// TIA Portal project "СУК 3.2 РАЕС-1.2 v1.1_20261002_1325" (V20)

(* hardware
DEVICE "S7-1500/ET200MP station_1"  S7-1500 station
   slot 0: "Rail_0"  Rack  6ES7 590-1***0-0AA0
   slot 1: "A1_1"  CPU 1515-2 PN  6ES7 515-2AN03-0AB0  V3.0
      slot 3: "CPU display_1"  6ES7591-1BA00-0AA0
      slot 32768: "PROFINET interface_1"  X1
         slot 32769: "Port_1"  X1 P1
         slot 32770: "Port_2"  X1 P2
      slot 33024: "PROFINET interface_2"  X2
         slot 33025: "Port_1"  X2 P1
      slot 34817: "Virtual CP interface port_1"  Virtual CP interface port  Virtual CP interface port
   slot 2: "A1_2"  DI 32x24VDC HF  6ES7 521-1BL00-0AB0  V2.2
   slot 3: "A1_3"  DI 32x24VDC HF  6ES7 521-1BL00-0AB0  V2.2
   slot 4: "A1_4"  AI 8xU/I HF  6ES7 531-7NF00-0AB0  V1.2
   slot 5: "A1_5"  DQ 16x24VDC/0.5A HF  6ES7 522-1BH01-0AB0  V1.0
DEVICE "A1_0"  TP700 Comfort
   slot 0: "A1_0"  TP700 Comfort  6AV2 124-0GC01-0AX0  17.0.0.0
   slot 1: "HMI_RT_1"  TP700 Comfort  6AV2 124-0GC01-0AX0  17.0.0.0
   slot 5: "A1_0.IE_CP_1"  PROFINET Interface  17.0.0.0
      slot 1: "PROFINET Interface_1"  PROFINET Interface
         slot 1: "Port_1"  Port
         slot 2: "Port_2"  Port
   slot 7: "A1_0.MPI/DP_CP_1"  MPI/DP Interface  17.0.0.0
DEVICE "SCALANCE XC-200"  SCALANCE X-Station
   slot 0: "SCALANCE X rack"  Rail
   slot 0: "A1.6"  SCALANCE XC208  6GK5 208-0BA00-2AC2  V4.4
DEVICE "GSD device_1"  GSD.Device.PN
   slot 0: "Rack"  Rack  V1.0
   slot 0: "1BR"  Multiturn 30 Bit V2.x  6FX2001-5*N25  V2.2.x
      slot 0: "MC-Encoder Multiturn 30 Bit"  MC-Encoder Multiturn 30 Bit
      slot 1: "PN-IO"  PN-IO
         slot 1: "Port 1"  Port 1
         slot 2: "Port 2"  Port 2
      slot 1: "EO Encoder Multiturn V2.x_1"  EO Encoder Multiturn V2.x
         slot 0: "Module Access Point"  Module Access Point
   slot 1: "Standard Telegram 89, PZD3/5"  Standard Telegram 89, PZD3/5
DEVICE "GSD device_2"  GSD.Device.PN
   slot 0: "Rack"  Rack  V1.0
   slot 0: "3BR"  Multiturn 30 Bit V2.x  6FX2001-5*N25  V2.2.x
      slot 0: "MC-Encoder Multiturn 30 Bit"  MC-Encoder Multiturn 30 Bit
      slot 1: "PN-IO"  PN-IO
         slot 1: "Port 1"  Port 1
         slot 2: "Port 2"  Port 2
      slot 1: "EO Encoder Multiturn V2.x_1"  EO Encoder Multiturn V2.x
         slot 0: "Module Access Point"  Module Access Point
   slot 1: "Standard Telegram 89, PZD3/5"  Standard Telegram 89, PZD3/5
DEVICE "GSD device_3"  GSD.Device.PN
   slot 0: "Rack"  Rack  V1.0
   slot 0: "4BR1"  Multiturn 30 Bit V2.x  6FX2001-5*N25  V2.2.x
      slot 0: "MC-Encoder Multiturn 30 Bit"  MC-Encoder Multiturn 30 Bit
      slot 1: "PN-IO"  PN-IO
         slot 1: "Port 1"  Port 1
         slot 2: "Port 2"  Port 2
      slot 1: "EO Encoder Multiturn V2.x_1"  EO Encoder Multiturn V2.x
         slot 0: "Module Access Point"  Module Access Point
   slot 1: "Standard Telegram 89, PZD3/5"  Standard Telegram 89, PZD3/5
DEVICE "GSD device_4"  GSD.Device.PN
   slot 0: "Rack"  Rack  V1.0
   slot 0: "4BR2"  Multiturn 30 Bit V2.x  6FX2001-5*N25  V2.2.x
      slot 0: "MC-Encoder Multiturn 30 Bit"  MC-Encoder Multiturn 30 Bit
      slot 1: "PN-IO"  PN-IO
         slot 1: "Port 1"  Port 1
         slot 2: "Port 2"  Port 2
      slot 1: "EO Encoder Multiturn V2.x_1"  EO Encoder Multiturn V2.x
         slot 0: "Module Access Point"  Module Access Point
   slot 1: "Standard Telegram 89, PZD3/5"  Standard Telegram 89, PZD3/5
DEVICE "SINAMICS S_1"  SINAMICS S120
   slot 0: "Drive unit_1"  S120 CU320-2 PN  6SL3040-1MA01-0Axx  V5.1
      slot 1: "PROFINET interface"  PROFINET
      slot 3: "Ethernet commissioning interface"  LAN
   slot 0: "U1"  S120 CU320-2 PN
   slot 1: "1UZ1"  PM
      slot 10: "Control Unit Adapter_1"  1UZ1  6SL3040-0PA00-0Axx
      slot 200: "Power Module_1"  1UZ1  6SL3210-1PE21-4UL0
      slot 1000: "1M1"  1UZ1  XMxxxxx-xxxxx-xxxx
   slot 2: "3UZ1"  PM
      slot 10: "Control Unit Adapter_1"  3UZ1  6SL3040-0PA00-0Axx
      slot 200: "Power Module_2"  3UZ1  6SL3210-1PE14-3UL1
      slot 1000: "3M1"  3UZ1  XMxxxxx-xxxxx-xxxx
   slot 3: "4UZ1"  PM
      slot 10: "Control Unit Adapter_1"  4UZ1  6SL3040-0PA00-0Axx
      slot 200: "Power Module_3"  4UZ1  6SL3210-1PE14-3UL1
      slot 1000: "4M1"  4UZ1  XMxxxxx-xxxxx-xxxx
   slot 4: "4UZ2"  PM
      slot 10: "Control Unit Adapter_1"  4UZ2  6SL3040-0PA00-0Axx
      slot 200: "Power Module_4"  4UZ2  6SL3210-1PE14-3UL1
      slot 1000: "4M2"  4UZ2  XMxxxxx-xxxxx-xxxx
*)

// ===== PLC "A1_1"  CPU 1515-2 PN =====

VAR_GLOBAL   // PLC tag table "Default tag table"
   "xInitMerker" AT %M3.0 : Bool;   // Ознака ініціалізація панелі
   "TestReset" AT %M0.0 : Bool;
   "Clock_Byte" AT %MB0 : Byte;
   "Clock_10Hz" AT %M0.0 : Bool;
   "Clock_5Hz" AT %M0.1 : Bool;
   "Clock_2.5Hz" AT %M0.2 : Bool;
   "Clock_2Hz" AT %M0.3 : Bool;
   "Clock_1.25Hz" AT %M0.4 : Bool;
   "Clock_1Hz" AT %M0.5 : Bool;
   "Clock_0.625Hz" AT %M0.6 : Bool;
   "Clock_0.5Hz" AT %M0.7 : Bool;
END_VAR

VAR_GLOBAL   // PLC tag table "IO_Tags"
   "6KM1" AT %I0.0 : Bool;   // Лінійний контактор включений
   "6KM2" AT %I0.1 : Bool;   // Контактор кіл управління 220В, 50Гц включений
   "6KV" AT %I0.2 : Bool;   // Контроль напруги введення, 380В, 50Гц
   "6SF5" AT %I0.3 : Bool;   // Вимикач кіл живлення обігріву 220В, 50Гц
   "6QF2" AT %I0.4 : Bool;   // Захист кіл гальм
   "6QF3" AT %I0.5 : Bool;   // Вимикач трансформатора 6Т1, 380В, 50Гц
   "6QF4" AT %I0.6 : Bool;   // Вимикач вторинних кіл трансформатора 6Т1, 380В, 50Гц
   "6SF1" AT %I0.7 : Bool;   // Вимикач живлення 6KV, 380В, 50Гц
   "6SF2" AT %I1.0 : Bool;   // Ввідний пристрій. Вимикач кіл управління 220В, 50Гц
   "6SF4" AT %I1.1 : Bool;   // Ввідний пристрій. Вимикач кіл живлення ОВП, 220В, 50Гц
   "6K3" AT %I1.2 : Bool;   // Ввідний пристрій. Команда на включення лінійного контактора з пульта
   "9QF2" AT %I1.3 : Bool;   // Вимикач трансформатора 9Т1, 380В, 50Гц
   "9QF3" AT %I1.4 : Bool;   // Вимикач ремонтного освітлення, 12В, 50Гц
   "9QF4" AT %I1.5 : Bool;   // Вимикач власних потреб шафа, 220В, 50Гц
   "9K2" AT %I1.6 : Bool;   // Контроль підігріву шафи SU1
   "9K3" AT %I1.7 : Bool;   // Сейсмодатчик
   "S1_Up" AT %I2.0 : Bool;   // Механізм підйому. Підйом 1-а швидкість
   "S1_Down" AT %I2.1 : Bool;   // Механізм підйому. Опускання 1-а швидкість
   "S1_Forward" AT %I2.2 : Bool;   // Механізм пересування візка. Вперед 1-а швидкість
   "S1_Backward" AT %I2.3 : Bool;   // Механізм пересування візка. Назад 1-а швидкість
   "S1_Left" AT %I2.4 : Bool;   // Механізм пересування крана. Вліво 1-а швидкість
   "S1_Right" AT %I2.5 : Bool;   // Механізм пересування крана. Управо 1-а швидкість
   "S2_Speed" AT %I2.6 : Bool;   // Перемикач 2-а швидкість
   "Bell" AT %I2.7 : Bool;   // Включення дзвінка
   "1BV" AT %I3.1 : Bool;   // Контроль обертання барабану
   "1BM1_Up" AT %I3.2 : Bool;   // Контроль роботи механізма підйому
   "1BM1_Brake" AT %I3.3 : Bool;   // Контроль зносу гальма механізму підйому
   "1K41" AT %I3.4 : Bool;   // Дозвіл роботи механізмупідйому. (РП роз'єданий з приводом)
   "4QF1" AT %I3.5 : Bool;   // Механізм пересування крана. Захист кіл гальм
   "4KT1" AT %I3.6 : Bool;   // Механізм пересування крана. Температурний захист двигуна 4M1
   "4KT2" AT %I3.7 : Bool;   // Механізм пересування крана. Температурний захист двигуна 4M2
   "1BT1" AT %I4.0 : Bool;   // Механізм підйому. Термозахист гальмівного резистора
   "1K1" AT %I4.1 : Bool;   // Механізм підйому. Дозвіл нормальної швидкості. Рух вгору
   "1K2" AT %I4.2 : Bool;   // Механізм підйому. Дозвіл нормальної швидкості. Рух вниз
   "1K3" AT %I4.3 : Bool;   // Механізм підйому. Дозвіл роботи. Рух вгору
   "1K4" AT %I4.4 : Bool;   // Механізм підйому. Дозвіл роботи. Рух вниз
   "1K11" AT %I4.5 : Bool;   // Механізм підйому. Перевищення номінального вантажу 115%
   "1K12" AT %I4.6 : Bool;   // Механізм підйому. Ослаблення канатів
   "1KT" AT %I4.7 : Bool;   // Механізм підйому. Температурний захист двигуна
   "1K21" AT %I5.0 : Bool;   // Механізм підйому. Вимикачі кінцеві на гальмі 1YB1. Гальмо розгальмоване
   "1K22" AT %I5.1 : Bool;   // Механізм підйому. Вимикачі кінцеві на гальмі 1YB1. Гальмо загальмоване
   "1K23" AT %I5.2 : Bool;   // Механізм підйому. Вимикачі кінцеві на гальмі 1YB1. Товщина гальмівних наладок в нормі
   "1K31" AT %I5.3 : Bool;   // Механізм підйому. Вимикачі кінцеві на гальмі 1YB2. Гальмо розгальмоване
   "1K32" AT %I5.4 : Bool;   // Механізм підйому. Вимикачі кінцеві на гальмі 1YB2. Гальмо загальмоване
   "1K33" AT %I5.5 : Bool;   // Механізм підйому. Вимикачі кінцеві на гальмі 1YB2. Дозвіл роботи (MPP роз'єднаний з гальмом)
   "1QF1" AT %I5.6 : Bool;   // Механізм підйому. Захист випрямляча гальма 1YB1
   "1QF2" AT %I5.7 : Bool;   // Механізм підйому. Захист випрямляча гальма 1YB2
   "3BT1" AT %I6.0 : Bool;   // Механізм пересування візка. Термозахист гальмівного резистора
   "3K1" AT %I6.1 : Bool;   // Механізм пересування візка. Дозвіл нормальної швидкості. Рух вперед
   "3K2" AT %I6.2 : Bool;   // Механізм пересування візка. Дозвіл роботи. Рух вперед
   "3K3" AT %I6.3 : Bool;   // Механізм пересування візка. Дозвіл нормальної швидкості. Рух назад
   "3K4" AT %I6.4 : Bool;   // Механізм пересування візка. Дозвіл роботи. Рух назад
   "3K41" AT %I6.5 : Bool;   // Механізм пересування візка. Дозвіл роботи (РП роз'єднан з приводом)
   "3KT" AT %I6.6 : Bool;   // Механізм пересування візка. Температурний захист двигуна
   "4K5" AT %I6.7 : Bool;   // Механізм пересування крана. Дозвіл роботи з будь-якої зі сторін від колони
   "4BT1" AT %I7.0 : Bool;   // Механізм пересування крана. Термозахист гальмівного резистора 4RT1
   "4BT2" AT %I7.1 : Bool;   // Механізм пересування крана. Термозахист гальмівного резистора 4RT2
   "4K1" AT %I7.2 : Bool;   // Механізм пересування крана. Дозвіл нормальної швидкості. Рух вліво
   "4K2" AT %I7.3 : Bool;   // Механізм пересування крана. Дозвіл нормальної швидкості. Рух управо
   "4K3" AT %I7.4 : Bool;   // Механізм пересування крана. Дозвіл роботи. Рух вліво
   "4K4" AT %I7.5 : Bool;   // Механізм пересування крана. Дозвіл роботи. Рух управо
   "4K41" AT %I7.6 : Bool;   // Механізм пересування крана. Дозвіл роботи (РП роз'єднан з приводом). 4SQ41
   "4K42" AT %I7.7 : Bool;   // Механізм пересування крана. Дозвіл роботи (РП роз'єднан з приводом). 4SQ42
   "1KM1" AT %Q0.0 : Bool;   // Включення рабочого гальма підйому
   "1KM2" AT %Q0.1 : Bool;   // Включення вбудованого гальма підйому
   "1KM3" AT %Q0.2 : Bool;   // Включення аварійного гальма підйому
   "3KM1" AT %Q0.3 : Bool;   // Включення рабочого гальма пересування візка
   "4KM1" AT %Q0.4 : Bool;   // Включення рабочих гальм пересування крана
   "6K1" AT %Q0.5 : Bool;   // Дозвіл включення лінійного контактора
   "6K2" AT %Q0.6 : Bool;   // Вимкнення лінійного контактора
   "9K1" AT %Q0.7 : Bool;   // Включення дзвінка
   "S1_1HL" AT %Q1.2 : Bool;   // Лампа. Готовність приводу підйому
   "S1_3HL" AT %Q1.3 : Bool;   // Лампа. Готовність приводу пересування візка
   "S1_4HL" AT %Q1.4 : Bool;   // Лампа. Готовність приводу пересування крана
   "S1_6HL1" AT %Q1.5 : Bool;   // Лампа. Лінійний контактор увімкнено
   "S1_6HL2" AT %Q1.6 : Bool;   // Лампа. Вхідна напруга не в нормі
   "1A1" AT %IW8 : Int;   // Контроль крутного моменту двигуна підйома
   "I3_0" AT %I3.0 : Bool;   // Резерв
   "IW10" AT %IW10 : Int;   // Резерв
   "IW12" AT %IW12 : Int;   // Резерв
   "IW14" AT %IW14 : Int;   // Резерв
   "IW16" AT %IW16 : Int;   // Резерв
   "IW18" AT %IW18 : Int;   // Резерв
   "IW20" AT %IW20 : Int;   // Резерв
   "IW22" AT %IW22 : Int;   // Резерв
   "Q1_0" AT %Q1.0 : Bool;   // Резерв
   "Q1_1" AT %Q1.1 : Bool;   // Резерв
   "Q1_7" AT %Q1.7 : Bool;   // Резерв
END_VAR

TYPE "udtMovePerm"
   STRUCT
      Upward : Bool;   // Дозвіл роботи. Рух вгору
      Downward : Bool;   // Дозвіл роботи. Рух вниз
      Forward : Bool;   // Дозвіл роботи. Рух вперед
      Backward : Bool;   // Дозвіл роботи. Рух назад
      Left : Bool;   // Дозвіл роботи. Рух вліво
      Right : Bool;   // Дозвіл роботи. Рух управо
      No_Pillar : Bool;   // Дозвіл роботи. Збудь-якої зі сторін від колони
   END_STRUCT;
END_TYPE

TYPE "DigICfg"
   STRUCT
      VRaw : Bool;   // RAW value
      Val : Bool;   // Value
      INV : Bool;   // Inverse raw value
      SVal : Bool;   // Value for simulation
      SML : Bool;   // Output value is simulated
      Text : WString;   // Tag name
      Chanal : WString;   // Chanal
   END_STRUCT;
END_TYPE

TYPE "udtMDM"
   STRUCT
      LM_WP_disconn_brake : Bool;   // Механізм підйому. Вимикачі кінцеві на гальмі 1YB2. Дозвіл роботи (MPP роз'єднаний з гальмом)
      LM_WP_disconn_drive : Bool;   // Механізм підйому. РП роз'єднаний з приводом
      TM_WP_disconn_drive : Bool;   // Механізм пересування візка. Дозвіл роботи (РП роз'єднан з приводом)
      CM_WP_disconn_drive_1 : Bool;   // Механізм пересування крана. Дозвіл роботи (РП роз'єднан з приводом). 4SQ41
      CM_WP_disconn_drive_2 : Bool;   // Механізм пересування крана. Дозвіл роботи (РП роз'єднан з приводом). 4SQ42
   END_STRUCT;
END_TYPE

TYPE "AnICfg"
   STRUCT
      VRaw : Int;   // Raw value (from input channel)
      LORaw : Int;   // Raw value LO limit
      HIRaw : Int;   // RAW value HI limit
      Val : Real;   // Output value
      LOEng : Real;   // Engineering (scaled) minimum value
      HIEng : Real;   // Engineering (scaled) maximum value
      FVal : Real;   // Filtered value
      PhyVal : Real;   // Physical value (mA)
      LOSP : Real;   // LO setpoint
      LOLOSP : Real;   // LO-LO setpoint
      HISP : Real;   // HI setpoint
      HIHISP : Real;   // HI-HI setpoint
      Hyst : Real;   // Hysteresis in real units
      SimVal : Real;   // Value for simulation
      LOEn : Bool;   // LO warning enabled
      LOLOEn : Bool;   // LO-LO Alarm enabled
      HIEn : Bool;   // HI warning enabled
      HIHIEn : Bool;   // HI-HI Alarm enabled
      LO : Bool;   // Low level is reached
      LOLO : Bool;   // Low Low level is reached
      HI : Bool;   // High level is reached
      HIHI : Bool;   // High High level is reached
      SML : Bool;   // Output value is simulated
      Reset : Bool;   // Reset
      STS : Int;   // Status
      T_FLTR : Int;   // Filtering time, x0.01 seconds
      Text : WString;   // Tag name
      Chanal : WString;   // Chanal
   END_STRUCT;
END_TYPE

TYPE "udtRemCtrl"
   STRUCT
      Btn_Up : Bool;   // 1SB1 Підйом 1 швидкість
      Btn_Down : Bool;   // 1SB2 Опускання 1 швидкість
      Btn_Fwd : Bool;   // 3SB1 Вперед 1-а швидкість
      Btn_Bwd : Bool;   // 3SB2 Назад 1-а швидкість
      Btn_Left : Bool;   // 4SB1 Управо 1-а швидкість
      Btn_Right : Bool;   // 4SB2 Вліво 1-а швидкість
      Btn_ScndSpeed : Bool;   // SB1 2 швидкість
      Btn_Bell : Bool;   // 9SB1 Включення дзвінка
   END_STRUCT;
END_TYPE

TYPE "DigOCfg"
   STRUCT
      VRaw : Bool;
      Val : Bool;
      SVal : Bool;
      SML : Bool;
      Text : WString;
      Chanal : WString;
   END_STRUCT;
END_TYPE

TYPE "udtSpeedPerm"
   STRUCT
      Speed_normal_Up : Bool;   // Дозвіл ном. швидкості вгору
      Speed_normal_Down : Bool;   // Дозвіл ном. швидкості вниз
      Speed_normal_Fwd : Bool;   // Дозвіл ном. швидкості вперед
      Speed_normal_Bwd : Bool;   // Дозвіл ном. швидкості назад
      Speed_normal_Left : Bool;   // Дозвіл ном. швидкості вліво
      Speed_normal_Right : Bool;   // Дозвіл ном. швидкості вправо
   END_STRUCT;
END_TYPE

// folder: Drives

TYPE "UDT_S120_Tel220_In"
   STRUCT
      ZSW1_BM : Word := W#16#0000;   // PZD1 Основне статусне слово ПЧ
      NIST_A : Int := 0;   // PZD2 Фактична швидкість
      IAIST : Int := 0;   // PZD3 Фактичний струм
      MIST : Int := 0;   // PZD4 Фактичний момент
      WARN_CODE : Word := W#16#0000;   // PZD5 Код попередження ПЧ
      FAULT_CODE : Word := W#16#0000;   // PZD6 Код аварії ПЧ
      ZSW2_BM : Word := W#16#0000;   // PZD7 Додаткове статусне слово ПЧ
      NSET_FB : Int := 0;   // PZD8 Зворотний зв'язок по завданню швидкості з ПЧ
      P_ACT : Int := 0;   // PZD9 Поточна активна потужність ПЧ
      BRAKE_STATUS : Word := W#16#0000;   // PZD10 Статус гальма з ПЧ, параметр r1229
   END_STRUCT;
END_TYPE

TYPE "UDT_S120_Tel220_Out"
   STRUCT
      STW1_BM : Word := W#16#0000;   // PZD1 Основне керуюче слово ПЧ
      NSOLL_B : DInt := 0;   // PZD2-PZD3 Завдання швидкості (32 Bits) / PZD2 Завдання швидкості
      STW2_BM : Word := W#16#0000;   // PZD4 Додаткове керуюче слово ПЧ / PZD3 Додаткове керуюче слово ПЧ
      M_ADD : Int := 0;   // PZD5 Додаткове завдання моменту / PZD4 Додаткове завдання моменту
      M_LIM : Int := 0;   // PZD6 Обмеження моменту / PZD5 Обмеження моменту
      USER_1 : Word := W#16#0000;   // PZD7 Резерв / сигнал прикладної логіки / PZD6 Резерв / сигнал прикладної логіки
      USER_2 : Word := W#16#0000;   // PZD8 Резерв / сигнал прикладної логіки / PZD7 Резерв / сигнал прикладної логіки
      USER_3 : Word := W#16#0000;   // PZD9 Резерв / сигнал прикладної логіки / PZD8 Резерв / сигнал прикладної логіки
      USER_4 : Word := W#16#0000;   // PZD10 Резерв / сигнал прикладної логіки / PZD9 Резерв / сигнал прикладної логіки
   END_STRUCT;
END_TYPE

TYPE "UDT_S120_BrakeStatus"
   STRUCT
      CommandOpenBrake : Bool := FALSE;   // Біт 01: команда відкрити гальмо, постійний сигнал
      PulseEnableExtendedBrakeControl : Bool := FALSE;   // Біт 03: імпульс дозволу розширеного керування гальмом
      BrakeDoesNotOpen : Bool := FALSE;   // Біт 04: гальмо не відкривається
      BrakeDoesNotClose : Bool := FALSE;   // Біт 05: гальмо не закривається
      BrakeThresholdExceeded : Bool := FALSE;   // Біт 06: перевищено поріг гальма
      BrakeThresholdUndershot : Bool := FALSE;   // Біт 07: значення нижче порогу гальма
      BrakeMonitoringTimeExpired : Bool := FALSE;   // Біт 08: перевищено час контролю гальма
      PulseEnableRequestMissing : Bool := FALSE;   // Біт 09: відсутній запит дозволу імпульсу / керування заблоковано
      BrakeOrLogicResult : Bool := FALSE;   // Біт 10: результат логіки OR для гальма
      BrakeAndLogicResult : Bool := FALSE;   // Біт 11: результат логіки AND для гальма
   END_STRUCT;
END_TYPE

TYPE "UDT_HMI_WordBits"
   STRUCT
      Bit00 : Bool := FALSE;   // Біт 00
      Bit01 : Bool := FALSE;   // Біт 01
      Bit02 : Bool := FALSE;   // Біт 02
      Bit03 : Bool := FALSE;   // Біт 03
      Bit04 : Bool := FALSE;   // Біт 04
      Bit05 : Bool := FALSE;   // Біт 05
      Bit06 : Bool := FALSE;   // Біт 06
      Bit07 : Bool := FALSE;   // Біт 07
      Bit08 : Bool := FALSE;   // Біт 08
      Bit09 : Bool := FALSE;   // Біт 09
      Bit10 : Bool := FALSE;   // Біт 10
      Bit11 : Bool := FALSE;   // Біт 11
      Bit12 : Bool := FALSE;   // Біт 12
      Bit13 : Bool := FALSE;   // Біт 13
      Bit14 : Bool := FALSE;   // Біт 14
      Bit15 : Bool := FALSE;   // Біт 15
   END_STRUCT;
END_TYPE

TYPE "UDT_HMI_S120_STW1"
   STRUCT
      OnOff1 : Bool := FALSE;   // Біт 00: ON / OFF1
      NoCoastStop : Bool := FALSE;   // Біт 01: OFF2 не активний
      NoQuickStop : Bool := FALSE;   // Біт 02: OFF3 / Quick Stop не активний
      EnableOperation : Bool := FALSE;   // Біт 03: дозвіл роботи ПЧ
      RampGeneratorEnable : Bool := FALSE;   // Біт 04: дозвіл генератора рампи
      RampGeneratorContinue : Bool := FALSE;   // Біт 05: продовження роботи генератора рампи
      SetpointEnable : Bool := FALSE;   // Біт 06: дозвіл завдання швидкості
      FaultAcknowledge : Bool := FALSE;   // Біт 07: квітування аварії ПЧ
      Reserved08 : Bool := FALSE;   // Біт 08: резерв / залежить від параметрування
      Reserved09 : Bool := FALSE;   // Біт 09: резерв / залежить від параметрування
      ControlByPLC : Bool := FALSE;   // Біт 10: керування від PLC
      Reserved11 : Bool := FALSE;   // Біт 11: резерв / залежить від параметрування
      Reserved12 : Bool := FALSE;   // Біт 12: резерв / залежить від параметрування
      Reserved13 : Bool := FALSE;   // Біт 13: резерв / залежить від параметрування
      Reserved14 : Bool := FALSE;   // Біт 14: резерв / залежить від параметрування
      Reserved15 : Bool := FALSE;   // Біт 15: резерв / залежить від параметрування
   END_STRUCT;
END_TYPE

TYPE "UDT_HMI_S120_ZSW1"
   STRUCT
      ReadyToSwitchOn : Bool := FALSE;   // Біт 00: ПЧ готовий до вмикання
      ReadyToOperate : Bool := FALSE;   // Біт 01: ПЧ готовий до роботи
      OperationEnabled : Bool := FALSE;   // Біт 02: робота ПЧ дозволена
      FaultActive : Bool := FALSE;   // Біт 03: активна аварія ПЧ
      NoCoastStopActive : Bool := FALSE;   // Біт 04: OFF2 не активний
      NoQuickStopActive : Bool := FALSE;   // Біт 05: OFF3 / Quick Stop не активний
      SwitchingOnInhibit : Bool := FALSE;   // Біт 06: активна заборона вмикання
      WarningActive : Bool := FALSE;   // Біт 07: активне попередження ПЧ
      SpeedErrorInTolerance : Bool := FALSE;   // Біт 08: відхилення швидкості в межах допуску / залежить від параметрування
      ControlRequested : Bool := FALSE;   // Біт 09: ПЧ запитує керування від PLC
      SetpointReached : Bool := FALSE;   // Біт 10: завдання досягнуто / залежить від параметрування
      InternalLimitActive : Bool := FALSE;   // Біт 11: активне внутрішнє обмеження
      Reserved12 : Bool := FALSE;   // Біт 12: резерв / залежить від параметрування
      Reserved13 : Bool := FALSE;   // Біт 13: резерв / залежить від параметрування
      Reserved14 : Bool := FALSE;   // Біт 14: резерв / залежить від параметрування
      Reserved15 : Bool := FALSE;   // Біт 15: резерв / залежить від параметрування
   END_STRUCT;
END_TYPE

TYPE "UDT_HMI_S120_BrakeStatus"
   STRUCT
      RawWord : Word := W#16#0000;   // Сире слово статусу гальма з ПЧ
      Bit00 : Bool := FALSE;   // Біт 00: резерв / не використовується
      CommandOpenBrake : Bool := FALSE;   // Біт 01: команда відкрити гальмо
      Bit02 : Bool := FALSE;   // Біт 02: резерв / не використовується
      PulseEnableExtendedBrakeControl : Bool := FALSE;   // Біт 03: імпульс дозволу розширеного керування гальмом
      BrakeDoesNotOpen : Bool := FALSE;   // Біт 04: гальмо не відкривається
      BrakeDoesNotClose : Bool := FALSE;   // Біт 05: гальмо не закривається
      BrakeThresholdExceeded : Bool := FALSE;   // Біт 06: перевищено поріг гальма
      BrakeThresholdUndershot : Bool := FALSE;   // Біт 07: значення нижче порогу гальма
      BrakeMonitoringTimeExpired : Bool := FALSE;   // Біт 08: перевищено час контролю гальма
      PulseEnableRequestMissing : Bool := FALSE;   // Біт 09: відсутній запит дозволу імпульсу / керування заблоковано
      BrakeOrLogicResult : Bool := FALSE;   // Біт 10: результат логіки OR для гальма
      BrakeAndLogicResult : Bool := FALSE;   // Біт 11: результат логіки AND для гальма
      Bit12 : Bool := FALSE;   // Біт 12: резерв / не використовується
      Bit13 : Bool := FALSE;   // Біт 13: резерв / не використовується
      Bit14 : Bool := FALSE;   // Біт 14: резерв / не використовується
      Bit15 : Bool := FALSE;   // Біт 15: резерв / не використовується
   END_STRUCT;
END_TYPE

TYPE "UDT_HMI_S120_RawTelegram"
   STRUCT
      STW1_BM : Word := W#16#0000;   // PZD1 PLC -> ПЧ: основне керуюче слово
      NSOLL_B : DInt := 0;   // PZD2-PZD3 PLC -> ПЧ: завдання швидкості (32 Bits) / PZD2 PLC -> ПЧ: завдання швидкості
      STW2_BM : Word := W#16#0000;   // PZD4 PLC -> ПЧ: додаткове керуюче слово / PZD3 PLC -> ПЧ: додаткове керуюче слово
      M_ADD : Int := 0;   // PZD5 PLC -> ПЧ: додаткове завдання моменту / PZD4 PLC -> ПЧ: додаткове завдання моменту
      M_LIM : Int := 0;   // PZD6 PLC -> ПЧ: обмеження моменту / PZD5 PLC -> ПЧ: обмеження моменту
      USER_1 : Word := W#16#0000;   // PZD7 PLC -> ПЧ: резерв / user PZD / PZD6 PLC -> ПЧ: резерв / user PZD
      USER_2 : Word := W#16#0000;   // PZD8 PLC -> ПЧ: резерв / user PZD / PZD7 PLC -> ПЧ: резерв / user PZD
      USER_3 : Word := W#16#0000;   // PZD9 PLC -> ПЧ: резерв / user PZD / PZD8 PLC -> ПЧ: резерв / user PZD
      USER_4 : Word := W#16#0000;   // PZD10 PLC -> ПЧ: резерв / user PZD / PZD9 PLC -> ПЧ: резерв / user PZD
      ZSW1_BM : Word := W#16#0000;   // PZD1 ПЧ -> PLC: основне статусне слово
      NIST_A : Int := 0;   // PZD2 ПЧ -> PLC: фактична швидкість
      IAIST : Int := 0;   // PZD3 ПЧ -> PLC: фактичний струм
      MIST : Int := 0;   // PZD4 ПЧ -> PLC: фактичний момент
      WARN_CODE : Word := W#16#0000;   // PZD5 ПЧ -> PLC: код попередження
      FAULT_CODE : Word := W#16#0000;   // PZD6 ПЧ -> PLC: код аварії
      ZSW2_BM : Word := W#16#0000;   // PZD7 ПЧ -> PLC: додаткове статусне слово
      NSET_FB : Int := 0;   // PZD8 ПЧ -> PLC: зворотний зв'язок завдання швидкості
      P_ACT : Int := 0;   // PZD9 ПЧ -> PLC: активна потужність
      BRAKE_STATUS : Word := W#16#0000;   // PZD10 ПЧ -> PLC: статус гальма
   END_STRUCT;
END_TYPE

TYPE "UDT_HMI_S120_Values"
   STRUCT
      AxisEnabled : Bool := FALSE;   // ПЧ увімкнений та робота дозволена
      Lockout : Bool := FALSE;   // ПЧ не готовий до роботи або активна блокування
      Error : Bool := FALSE;   // Помилка драйвера або аварія ПЧ
      BrakeOpenRequest : Bool := FALSE;   // ПЧ запитує відкриття гальма
      ActVelocity_Rpm : Real := 0.0;   // Фактична швидкість, об/хв
      SpeedSetpointFb_Rpm : Real := 0.0;   // Зворотний зв'язок по завданню швидкості, об/хв
      ActCurrent_A : Real := 0.0;   // Фактичний струм, А
      ActTorque_Nm : Real := 0.0;   // Фактичний момент, Н·м
      ActPower_kW : Real := 0.0;   // Поточна активна потужність, кВт
      LoadPower_Pct : Real := 0.0;   // Завантаження по потужності, %
      FaultCode : Word := W#16#0000;   // Код аварії ПЧ
      WarningCode : Word := W#16#0000;   // Код попередження ПЧ
      Status : Word := W#16#0000;   // Статус драйвера, бітове слово
      DiagId : Word := W#16#0000;   // Код діагностики драйвера
      SpeedError_Rpm : Real := 0.0;   // Помилка по швидкості (різниця SP-FB), об/хв
   END_STRUCT;
END_TYPE

TYPE "UDT_HMI_S120_Drive"
   STRUCT
      Values : "UDT_HMI_S120_Values";   // Основні значення та діагностика ПЧ
      StatusBits : "UDT_HMI_S120_DriverStatus";   // Біти статусу драйвера ПЧ
      Raw : "UDT_HMI_S120_RawTelegram";   // Сирі дані telegram 220
      STW1 : "UDT_HMI_S120_STW1";   // Біти керуючого слова STW1_BM
      STW2 : "UDT_HMI_WordBits";   // Біти додаткового керуючого слова STW2_BM
      ZSW1 : "UDT_HMI_S120_ZSW1";   // Біти основного статусного слова ZSW1_BM
      ZSW2 : "UDT_HMI_WordBits";   // Біти додаткового статусного слова ZSW2_BM
      Brake : "UDT_HMI_S120_BrakeStatus";   // Біти статусу гальма з ПЧ
      Faults : Struct   // Помилки ПЧ (для алармів)
         FaultsWord1 : Word;   // Слово помилок 1
         FaultsWord2 : Word;   // Слово помилок 2
         FaultsWord3 : Word;   // Слово помилок 3
         FaultsWord4 : Word;   // Слово помилок 4
      END_STRUCT;
      Alarms : Struct   // Помилки ПЧ (для алармів) / Попередження ПЧ (для алармів)
         AlarmsWord1 : Word;   // Слово попереджень 1
         AlarmsWord2 : Word;   // Слово попереджень 2
         AlarmsWord3 : Word;   // Слово попереджень 3
         AlarmsWord4 : Word;   // Слово попереджень 4
      END_STRUCT;
   END_STRUCT;
END_TYPE

TYPE "UDT_HMI_S120_DriverStatus"
   STRUCT
      ReadOk : Bool := FALSE;   // Біт 00: читання telegram ПЧ -> PLC виконано без помилки
      WriteOk : Bool := FALSE;   // Біт 01: запис telegram PLC -> ПЧ виконано без помилки
      AxisEnabled : Bool := FALSE;   // Біт 02: ПЧ увімкнений та робота дозволена
      Lockout : Bool := FALSE;   // Біт 03: ПЧ не готовий до роботи або активна блокування
      DriveFault : Bool := FALSE;   // Біт 04: аварія ПЧ активна
      DriveWarning : Bool := FALSE;   // Біт 05: попередження ПЧ активне
      BrakeOpenRequest : Bool := FALSE;   // Біт 06: ПЧ запитує відкриття гальма
      SimMode : Bool := FALSE;   // Біт 07: активний режим симуляції
      SwitchingOnInhibit : Bool := FALSE;   // Біт 08: активна заборона вмикання
      ControlRequested : Bool := FALSE;   // Біт 09: ПЧ запитує керування від PLC
      Reserved10 : Bool := FALSE;   // Біт 10: резерв
      Reserved11 : Bool := FALSE;   // Біт 11: резерв
      Reserved12 : Bool := FALSE;   // Біт 12: резерв
      Reserved13 : Bool := FALSE;   // Біт 13: резерв
      Reserved14 : Bool := FALSE;   // Біт 14: резерв
      Reserved15 : Bool := FALSE;   // Біт 15: резерв
   END_STRUCT;
END_TYPE

// folder: Drives/Tlg390_CU

TYPE "UDT_S120_Tel390_CU_In"
   STRUCT
      CU_ZSW1 : Word := W#16#0000;   // PZD1 Статусне слово CU320-2 PN
      CU_DIAG_CODE : Word := W#16#0000;   // PZD2 Діагностичне слово / код помилки або попередження CU
   END_STRUCT;
END_TYPE

TYPE "UDT_S120_Tel390_CU_Out"
   STRUCT
      CU_STW1 : Word := W#16#0000;   // PZD1 Керуюче слово CU320-2 PN
      CU_CTRL2 : Word := W#16#0000;   // PZD2 Резерв / службове слово PLC -> CU
   END_STRUCT;
END_TYPE

TYPE "UDT_S120_Tel390_CU_ZSW1_Bits"
   STRUCT
      ReadyToSwitchOn : Bool := FALSE;   // Біт 00: CU готова до вмикання / готовність
      ReadyToOperate : Bool := FALSE;   // Біт 01: CU готова до роботи
      OperationEnabled : Bool := FALSE;   // Біт 02: робота дозволена / стан OK
      FaultActive : Bool := FALSE;   // Біт 03: активна помилка CU
      NoCoastStopActive : Bool := FALSE;   // Біт 04: OFF2 не активний, якщо застосовується
      NoQuickStopActive : Bool := FALSE;   // Біт 05: OFF3 не активний, якщо застосовується
      SwitchingOnInhibit : Bool := FALSE;   // Біт 06: активна заборона вмикання / блокування
      WarningActive : Bool := FALSE;   // Біт 07: активне попередження CU
      Bit08 : Bool := FALSE;   // Біт 08: стан CU, залежить від параметрування
      ControlRequested : Bool := FALSE;   // Біт 09: CU запитує керування від PLC, якщо застосовується
      Bit10 : Bool := FALSE;   // Біт 10: стан CU, залежить від параметрування
      Bit11 : Bool := FALSE;   // Біт 11: стан CU, залежить від параметрування
      Bit12 : Bool := FALSE;   // Біт 12: стан CU, залежить від параметрування
      Bit13 : Bool := FALSE;   // Біт 13: стан CU, залежить від параметрування
      Bit14 : Bool := FALSE;   // Біт 14: стан CU, залежить від параметрування
      Bit15 : Bool := FALSE;   // Біт 15: стан CU, залежить від параметрування
   END_STRUCT;
END_TYPE

TYPE "UDT_HMI_S120_CU_Values"
   STRUCT
      CommOk : Bool := FALSE;   // Обмін з CU справний
      Fault : Bool := FALSE;   // CU повідомляє активну помилку
      Warning : Bool := FALSE;   // CU повідомляє активне попередження
      Error : Bool := FALSE;   // Помилка драйвера, комунікації або fault CU
      CU_StatusWord : Word := W#16#0000;   // Сире статусне слово CU, PZD1
      CU_DiagCode : Word := W#16#0000;   // Діагностичне слово / код помилки або попередження CU, PZD2
      Status : Word := W#16#0000;   // Статус драйвера CU, бітове слово
      DiagId : Word := W#16#0000;   // Код діагностики драйвера CU
   END_STRUCT;
END_TYPE

TYPE "UDT_HMI_S120_CU_RawTelegram"
   STRUCT
      CU_STW1 : Word := W#16#0000;   // PZD1 PLC -> CU: керуюче слово CU_STW1
      CU_CTRL2 : Word := W#16#0000;   // PZD2 PLC -> CU: резерв / службове слово
      CU_ZSW1 : Word := W#16#0000;   // PZD1 CU -> PLC: статусне слово CU_ZSW1
      CU_DIAG_CODE : Word := W#16#0000;   // PZD2 CU -> PLC: діагностичне слово / код
   END_STRUCT;
END_TYPE

TYPE "UDT_HMI_S120_CU_STW1"
   STRUCT
      Bit00 : Bool := FALSE;   // Біт 00: резерв / залежить від параметрування
      Bit01 : Bool := FALSE;   // Біт 01: резерв / залежить від параметрування
      Bit02 : Bool := FALSE;   // Біт 02: резерв / залежить від параметрування
      Bit03 : Bool := FALSE;   // Біт 03: резерв / залежить від параметрування
      Bit04 : Bool := FALSE;   // Біт 04: резерв / залежить від параметрування
      Bit05 : Bool := FALSE;   // Біт 05: резерв / залежить від параметрування
      Bit06 : Bool := FALSE;   // Біт 06: резерв / залежить від параметрування
      FaultAcknowledge : Bool := FALSE;   // Біт 07: квітування помилки CU
      Bit08 : Bool := FALSE;   // Біт 08: резерв / залежить від параметрування
      Bit09 : Bool := FALSE;   // Біт 09: резерв / залежить від параметрування
      RemoteControlByPLC : Bool := FALSE;   // Біт 10: Remote control / Master control by PLC
      Bit11 : Bool := FALSE;   // Біт 11: резерв / залежить від параметрування
      Bit12 : Bool := FALSE;   // Біт 12: резерв / залежить від параметрування
      Bit13 : Bool := FALSE;   // Біт 13: резерв / залежить від параметрування
      Bit14 : Bool := FALSE;   // Біт 14: резерв / залежить від параметрування
      Bit15 : Bool := FALSE;   // Біт 15: резерв / залежить від параметрування
   END_STRUCT;
END_TYPE

TYPE "UDT_HMI_S120_CU_ZSW1"
   STRUCT
      ReadyToSwitchOn : Bool := FALSE;   // Біт 00: CU готова до вмикання / готовність
      ReadyToOperate : Bool := FALSE;   // Біт 01: CU готова до роботи
      OperationEnabled : Bool := FALSE;   // Біт 02: робота дозволена / стан OK
      FaultActive : Bool := FALSE;   // Біт 03: активна помилка CU
      NoCoastStopActive : Bool := FALSE;   // Біт 04: OFF2 не активний, якщо застосовується
      NoQuickStopActive : Bool := FALSE;   // Біт 05: OFF3 не активний, якщо застосовується
      SwitchingOnInhibit : Bool := FALSE;   // Біт 06: активна заборона вмикання / блокування
      WarningActive : Bool := FALSE;   // Біт 07: активне попередження CU
      Bit08 : Bool := FALSE;   // Біт 08: стан CU, залежить від параметрування
      ControlRequested : Bool := FALSE;   // Біт 09: CU запитує керування від PLC
      Bit10 : Bool := FALSE;   // Біт 10: стан CU, залежить від параметрування
      Bit11 : Bool := FALSE;   // Біт 11: стан CU, залежить від параметрування
      Bit12 : Bool := FALSE;   // Біт 12: стан CU, залежить від параметрування
      Bit13 : Bool := FALSE;   // Біт 13: стан CU, залежить від параметрування
      Bit14 : Bool := FALSE;   // Біт 14: стан CU, залежить від параметрування
      Bit15 : Bool := FALSE;   // Біт 15: стан CU, залежить від параметрування
   END_STRUCT;
END_TYPE

TYPE "UDT_HMI_S120_CU_DriverStatus"
   STRUCT
      ReadOk : Bool := FALSE;   // Біт 00: читання telegram CU -> PLC виконано без помилки
      WriteOk : Bool := FALSE;   // Біт 01: запис telegram PLC -> CU виконано без помилки
      CommOk : Bool := FALSE;   // Біт 02: обмін з CU справний
      Fault : Bool := FALSE;   // Біт 03: fault CU
      Warning : Bool := FALSE;   // Біт 04: warning CU
      SwitchingOnInhibit : Bool := FALSE;   // Біт 05: заборона / блокування CU
      ControlRequested : Bool := FALSE;   // Біт 06: CU запитує керування від PLC
      SimMode : Bool := FALSE;   // Біт 07: активний режим симуляції
      Reserved08 : Bool := FALSE;   // Біт 08: резерв
      Reserved09 : Bool := FALSE;   // Біт 09: резерв
      Reserved10 : Bool := FALSE;   // Біт 10: резерв
      Reserved11 : Bool := FALSE;   // Біт 11: резерв
      Reserved12 : Bool := FALSE;   // Біт 12: резерв
      Reserved13 : Bool := FALSE;   // Біт 13: резерв
      Reserved14 : Bool := FALSE;   // Біт 14: резерв
      Reserved15 : Bool := FALSE;   // Біт 15: резерв
   END_STRUCT;
END_TYPE

TYPE "UDT_HMI_S120_CU"
   STRUCT
      Values : "UDT_HMI_S120_CU_Values";   // Основні значення та діагностика CU
      StatusBits : "UDT_HMI_S120_CU_DriverStatus";   // Біти статусу драйвера CU
      Raw : "UDT_HMI_S120_CU_RawTelegram";   // Сирі дані telegram 390
      STW1 : "UDT_HMI_S120_CU_STW1";   // Біти керуючого слова CU_STW1
      ZSW1 : "UDT_HMI_S120_CU_ZSW1";   // Біти статусного слова CU_ZSW1
   END_STRUCT;
END_TYPE

// folder: Encoders

TYPE "UDT_Enc_Tlg89_Out"
   STRUCT
      STW2_ENC : Word;   // Control word від PLC до енкодера.
      G1_XIST_PRESET_B1 : DInt;   // Значення preset для Telegram 89.
   END_STRUCT;
END_TYPE

TYPE "UDT_Enc_Tlg89_In"
   STRUCT
      ZSW2_ENC : Word;   // Status word енкодера.
      G1_XIST2 : DInt;   // Абсолютне положення енкодера.
      NIST_B : DInt;   // Фактична швидкість енкодера.
   END_STRUCT;
END_TYPE

TYPE "UDT_HMI_Encoder_View"
   STRUCT
      RawPosition : DInt := 0;   // Поточне raw-положення енкодера з G1_XIST2.
      RawVelocity : DInt := 0;   // Поточна raw-швидкість енкодера з NIST_B.
      EncoderReady : Bool := FALSE;   // Енкодер готовий для використання в логіці.
      PositionDataValid : Bool := FALSE;   // Положення енкодера достовірне.
      VelocityDataValid : Bool := FALSE;   // Швидкість енкодера достовірна.
      CommunicationFault : Bool := FALSE;   // Загальна помилка обміну з енкодером.
      EncoderFault : Bool := FALSE;   // Активна помилка енкодера.
      ErrorCode : DInt := DINT#0;   // Код активної помилки енкодера. 0 - помилки немає.
      EncoderAlarm : Bool := FALSE;   // Попередження енкодера.
      EncoderLifeValid : Bool := FALSE;   // Sign-of-life енкодера валідний.
      PresetBusy : Bool := FALSE;   // Preset-процедура активна.
      PresetDone : Bool := FALSE;   // Preset успішно виконано.
      PresetError : Bool := FALSE;   // Помилка виконання preset.
      PresetStatus : Word := 16#0000;   // Діагностичний код preset-процедури.
      STW2_ENC : Word := 16#0000;   // Control word Telegram 89 від PLC до енкодера.
      ZSW2_ENC : Word := 16#0000;   // Status word Telegram 89 від енкодера до PLC.
      Status : Word := 16#0000;   // Загальне діагностичне слово комунікаційного FB.
      Position_mm : Real := 0.0;   // Поточне масштабоване положення механізму, мм
      PositionRounded_mm : DInt := 0;   // Поточне округлене масштабоване положення механізму, мм
      PositionValid : Bool := FALSE;   // TRUE = масштабоване положення достовірне
   END_STRUCT;
END_TYPE

// folder: InOut

TYPE "udtInputCfg"
   STRUCT
      DigIn_0_0 : "DigICfg";   // Лінійний контактор включений
      DigIn_0_1 : "DigICfg";   // Контактор кіл управління 220В, 50Гц включений
      DigIn_0_2 : "DigICfg";   // Контроль напруги введення, 380В, 50Гц
      DigIn_0_3 : "DigICfg";   // Вимикач кіл живлення обігріву 220В, 50Гц
      DigIn_0_4 : "DigICfg";   // Захист кіл гальм
      DigIn_0_5 : "DigICfg";   // Вимикач трансформатора 6Т1, 380В, 50Гц
      DigIn_0_6 : "DigICfg";   // Вимикач вторинних кіл трансформатора 6Т1, 380В, 50Гц
      DigIn_0_7 : "DigICfg";   // Вимикач живлення 6KV, 380В, 50Гц
      DigIn_1_0 : "DigICfg";   // Ввідний пристрій. Вимикач кіл управління 220В, 50Гц
      DigIn_1_1 : "DigICfg";   // Ввідний пристрій. Вимикач кіл живлення ОВП, 220В, 50Гц
      DigIn_1_2 : "DigICfg";   // Ввідний пристрій. Команда на включення лінійного контактора з пульта
      DigIn_1_3 : "DigICfg";   // Вимикач трансформатора 9Т1, 380В, 50Гц
      DigIn_1_4 : "DigICfg";   // Вимикач ремонтного освітлення, 12В, 50Гц
      DigIn_1_5 : "DigICfg";   // Вимикач власних потреб шафа, 220В, 50Гц
      DigIn_1_6 : "DigICfg";   // Контроль підігріву шафи SU1
      DigIn_1_7 : "DigICfg";   // Сейсмодатчик
      DigIn_2_0 : "DigICfg";   // Механізм підйому. Підйом 1-а швидкість
      DigIn_2_1 : "DigICfg";   // Механізм підйому. Опускання 1-а швидкість
      DigIn_2_2 : "DigICfg";   // Механізм пересування візка. Вперед 1-а швидкість
      DigIn_2_3 : "DigICfg";   // Механізм пересування візка. Назад 1-а швидкість
      DigIn_2_4 : "DigICfg";   // Механізм пересування крана. Вліво 1-а швидкість
      DigIn_2_5 : "DigICfg";   // Механізм пересування крана. Управо 1-а швидкість
      DigIn_2_6 : "DigICfg";   // 2-а швидкість
      DigIn_2_7 : "DigICfg";   // Включення дзвінка
      DigIn_3_0 : "DigICfg";   // Spare / Резерв
      DigIn_3_1 : "DigICfg";   // Контроль обертання барабану
      DigIn_3_2 : "DigICfg";   // Контроль роботи механізма підйому
      DigIn_3_3 : "DigICfg";   // Контроль зносу гальма механізма підйому
      DigIn_3_4 : "DigICfg";   // Дозвіл роботи механізму підйому. (РП роз'єданий з приводом)
      DigIn_3_5 : "DigICfg";   // Механізм пересування крана. Захист кіл гальм
      DigIn_3_6 : "DigICfg";   // Механізм пересування крана. Температурний захист двигуна 4M1
      DigIn_3_7 : "DigICfg";   // Механізм пересування крана. Температурний захист двигуна 4M2
      DigIn_4_0 : "DigICfg";   // Механізм підйому. Термозахист гальмівного резистора
      DigIn_4_1 : "DigICfg";   // Механізм підйому. Дозвіл нормальної швидкості. Рух вгору
      DigIn_4_2 : "DigICfg";   // Механізм підйому. Дозвіл нормальної швидкості. Рух вниз
      DigIn_4_3 : "DigICfg";   // Механізм підйому. Дозвіл роботи. Рух вгору
      DigIn_4_4 : "DigICfg";   // Механізм підйому. Дозвіл роботи. Рух вниз
      DigIn_4_5 : "DigICfg";   // Механізм підйому. Перевищення номінального вантажу 115%
      DigIn_4_6 : "DigICfg";   // Механізм підйому. Ослаблення канатів
      DigIn_4_7 : "DigICfg";   // Механізм підйому. Температурний захист двигуна
      DigIn_5_0 : "DigICfg";   // Механізм підйому. Вимикачі кінцеві на гальмі 1YB1. Гальмо розгальмоване
      DigIn_5_1 : "DigICfg";   // Механізм підйому. Вимикачі кінцеві на гальмі 1YB1. Гальмо загальмоване
      DigIn_5_2 : "DigICfg";   // Механізм підйому. Вимикачі кінцеві на гальмі 1YB1. Товщина гальмівних наладок в нормі
      DigIn_5_3 : "DigICfg";   // Механізм підйому. Вимикачі кінцеві на гальмі 1YB2. Гальмо розгальмоване
      DigIn_5_4 : "DigICfg";   // Механізм підйому. Вимикачі кінцеві на гальмі 1YB2. Гальмо загальмоване
      DigIn_5_5 : "DigICfg";   // Механізм підйому. Вимикачі кінцеві на гальмі 1YB2. Дозвіл роботи (MPP роз'єднаний з гальмом)
      DigIn_5_6 : "DigICfg";   // Механізм підйому. Захист випрямляча гальма 1YB1
      DigIn_5_7 : "DigICfg";   // Механізм підйому. Захист випрямляча гальма 1YB2
      DigIn_6_0 : "DigICfg";   // Механізм пересування візка. Термозахист гальмівного резистора
      DigIn_6_1 : "DigICfg";   // Механізм пересування візка. Дозвіл нормальної швидкості. Рух вперед
      DigIn_6_2 : "DigICfg";   // Механізм пересування візка. Дозвіл роботи. Рух вперед
      DigIn_6_3 : "DigICfg";   // Механізм пересування візка. Дозвіл нормальної швидкості. Рух назад
      DigIn_6_4 : "DigICfg";   // Механізм пересування візка. Дозвіл роботи. Рух назад
      DigIn_6_5 : "DigICfg";   // Механізм пересування візка. Дозвіл роботи (РП роз'єднан з приводом)
      DigIn_6_6 : "DigICfg";   // Механізм пересування візка. Температурний захист двигуна
      DigIn_6_7 : "DigICfg";   // Механізм пересування крана. Дозвіл роботи з будь-якої зі сторін від колони
      DigIn_7_0 : "DigICfg";   // Механізм пересування крана. Термозахист гальмівного резистора 4RT1
      DigIn_7_1 : "DigICfg";   // Механізм пересування крана. Термозахист гальмівного резистора 4RT2
      DigIn_7_2 : "DigICfg";   // Механізм пересування крана. Дозвіл нормальної швидкості. Рух вліво
      DigIn_7_3 : "DigICfg";   // Механізм пересування крана. Дозвіл нормальної швидкості. Рух управо
      DigIn_7_4 : "DigICfg";   // Механізм пересування крана. Дозвіл роботи. Рух вліво
      DigIn_7_5 : "DigICfg";   // Механізм пересування крана. Дозвіл роботи. Рух управо
      DigIn_7_6 : "DigICfg";   // Механізм пересування крана. Дозвіл роботи (РП роз'єднан з приводом). 4SQ41
      DigIn_7_7 : "DigICfg";   // Механізм пересування крана. Дозвіл роботи (РП роз'єднан з приводом). 4SQ42
   END_STRUCT;
   // DigIn_0_0.Text := WSTRING#'Лінійний контактор включений';
   // DigIn_0_0.Chanal := WSTRING#'0';
   // DigIn_0_1.Text := WSTRING#'Контактор кіл управління 220В, 50Гц включений';
   // DigIn_0_1.Chanal := WSTRING#'1';
   // DigIn_0_2.Text := WSTRING#'Контроль напруги введення, 380В, 50Гц';
   // DigIn_0_2.Chanal := WSTRING#'2';
   // DigIn_0_3.Text := WSTRING#'Вимикач кіл живлення обігріву 220В, 50Гц';
   // DigIn_0_3.Chanal := WSTRING#'3';
   // DigIn_0_4.Text := WSTRING#'Захист кіл гальм';
   // DigIn_0_4.Chanal := WSTRING#'4';
   // DigIn_0_5.Text := WSTRING#'Вимикач трансформатора 6Т1, 380В, 50Гц';
   // DigIn_0_5.Chanal := WSTRING#'5';
   // DigIn_0_6.Text := WSTRING#'Вимикач вторинних кіл трансформатора 6Т1, 380В, 50Гц';
   // DigIn_0_6.Chanal := WSTRING#'6';
   // DigIn_0_7.Text := WSTRING#'Вимикач живлення 6KV, 380В, 50Гц';
   // DigIn_0_7.Chanal := WSTRING#'7';
   // DigIn_1_0.Text := WSTRING#'Ввідний пристрій. Вимикач кіл управління 220В, 50Гц';
   // DigIn_1_0.Chanal := WSTRING#'8';
   // DigIn_1_1.Text := WSTRING#'Ввідний пристрій. Вимикач кіл живлення ОВП, 220В, 50Гц';
   // DigIn_1_1.Chanal := WSTRING#'9';
   // DigIn_1_2.Text := WSTRING#'Ввідний пристрій. Команда на включення лінійного контактора з пульта';
   // DigIn_1_2.Chanal := WSTRING#'10';
   // DigIn_1_3.Text := WSTRING#'Вимикач трансформатора 9Т1, 380В, 50Гц';
   // DigIn_1_3.Chanal := WSTRING#'11';
   // DigIn_1_4.Text := WSTRING#'Вимикач ремонтного освітлення, 12В, 50Гц';
   // DigIn_1_4.Chanal := WSTRING#'12';
   // DigIn_1_5.Text := WSTRING#'Вимикач власних потреб шафа, 220В, 50Гц';
   // DigIn_1_5.Chanal := WSTRING#'13';
   // DigIn_1_6.Text := WSTRING#'Контроль підігріву шафи SU1';
   // DigIn_1_6.Chanal := WSTRING#'14';
   // DigIn_1_7.Text := WSTRING#'Сейсмодатчик';
   // DigIn_1_7.Chanal := WSTRING#'15';
   // DigIn_2_0.Text := WSTRING#'Механізм підйому. Підйом 1-а швидкість';
   // DigIn_2_0.Chanal := WSTRING#'16';
   // DigIn_2_1.Text := WSTRING#'Механізм підйому. Опускання 1-а швидкість';
   // DigIn_2_1.Chanal := WSTRING#'17';
   // DigIn_2_2.Text := WSTRING#'Механізм пересування візка. Вперед 1-а швидкість';
   // DigIn_2_2.Chanal := WSTRING#'18';
   // DigIn_2_3.Text := WSTRING#'Механізм пересування візка. Назад 1-а швидкість';
   // DigIn_2_3.Chanal := WSTRING#'19';
   // DigIn_2_4.Text := WSTRING#'Механізм пересування крана. Вліво 1-а швидкість';
   // DigIn_2_4.Chanal := WSTRING#'20';
   // DigIn_2_5.Text := WSTRING#'Механізм пересування крана. Управо 1-а швидкість';
   // DigIn_2_5.Chanal := WSTRING#'21';
   // DigIn_2_6.Text := WSTRING#'2-а швидкість';
   // DigIn_2_6.Chanal := WSTRING#'22';
   // DigIn_2_7.Text := WSTRING#'Включення дзвінка';
   // DigIn_2_7.Chanal := WSTRING#'23';
   // DigIn_3_0.Text := WSTRING#'Резерв';
   // DigIn_3_0.Chanal := WSTRING#'24';
   // DigIn_3_1.Text := WSTRING#'Контроль обертання барабану';
   // DigIn_3_1.Chanal := WSTRING#'25';
   // DigIn_3_2.Text := WSTRING#'Контроль роботи механізма підйому';
   // DigIn_3_2.Chanal := WSTRING#'26';
   // DigIn_3_3.Text := WSTRING#'Контроль зносу гальма механізма підйому';
   // DigIn_3_3.Chanal := WSTRING#'27';
   // DigIn_3_4.Text := WSTRING#'Дозвіл роботи механізму підйому. (РП розєданий з приводом)';
   // DigIn_3_4.Chanal := WSTRING#'28';
   // DigIn_3_5.Text := WSTRING#'Механізм пересування крана. Захист кіл гальм';
   // DigIn_3_5.Chanal := WSTRING#'29';
   // DigIn_3_6.Text := WSTRING#'Механізм пересування крана. Температурний захист двигуна 4M1';
   // DigIn_3_6.Chanal := WSTRING#'30';
   // DigIn_3_7.Text := WSTRING#'Механізм пересування крана. Температурний захист двигуна 4M2';
   // DigIn_3_7.Chanal := WSTRING#'31';
   // DigIn_4_0.Text := WSTRING#'Механізм підйому. Термозахист гальмівного резистора';
   // DigIn_4_0.Chanal := WSTRING#'0';
   // DigIn_4_1.Text := WSTRING#'Механізм підйому. Дозвіл нормальної швидкості. Рух вгору';
   // DigIn_4_1.Chanal := WSTRING#'1';
   // DigIn_4_2.Text := WSTRING#'Механізм підйому. Дозвіл нормальної швидкості. Рух вниз';
   // DigIn_4_2.Chanal := WSTRING#'2';
   // DigIn_4_3.Text := WSTRING#'Механізм підйому. Дозвіл роботи. Рух вгору';
   // DigIn_4_3.Chanal := WSTRING#'3';
   // DigIn_4_4.Text := WSTRING#'Механізм підйому. Дозвіл роботи. Рух вниз';
   // DigIn_4_4.Chanal := WSTRING#'4';
   // DigIn_4_5.Text := WSTRING#'Механізм підйому. Перевищення номінального вантажу 115%';
   // DigIn_4_5.Chanal := WSTRING#'5';
   // DigIn_4_6.Text := WSTRING#'Механізм підйому. Ослаблення канатів';
   // DigIn_4_6.Chanal := WSTRING#'6';
   // DigIn_4_7.Text := WSTRING#'Механізм підйому. Температурний захист двигуна';
   // DigIn_4_7.Chanal := WSTRING#'7';
   // DigIn_5_0.Text := WSTRING#'Механізм підйому. Вимикачі кінцеві на гальмі 1YB1. Гальмо розгальмоване';
   // DigIn_5_0.Chanal := WSTRING#'8';
   // DigIn_5_1.Text := WSTRING#'Механізм підйому. Вимикачі кінцеві на гальмі 1YB1. Гальмо загальмоване';
   // DigIn_5_1.Chanal := WSTRING#'9';
   // DigIn_5_2.Text := WSTRING#'Механізм підйому. Вимикачі кінцеві на гальмі 1YB1. Товщина гальмівних наладок в нормі';
   // DigIn_5_2.Chanal := WSTRING#'10';
   // DigIn_5_3.Text := WSTRING#'Механізм підйому. Вимикачі кінцеві на гальмі 1YB2. Гальмо розгальмоване';
   // DigIn_5_3.Chanal := WSTRING#'11';
   // DigIn_5_4.Text := WSTRING#'Механізм підйому. Вимикачі кінцеві на гальмі 1YB2. Гальмо загальмоване';
   // DigIn_5_4.Chanal := WSTRING#'12';
   // DigIn_5_5.Text := WSTRING#'Механізм підйому. Вимикачі кінцеві на гальмі 1YB2. Дозвіл роботи (MPP розєднаний з гальмом)';
   // DigIn_5_5.Chanal := WSTRING#'13';
   // DigIn_5_6.Text := WSTRING#'Механізм підйому. Захист випрямляча гальма 1YB1';
   // DigIn_5_6.Chanal := WSTRING#'14';
   // DigIn_5_7.Text := WSTRING#'Механізм підйому. Захист випрямляча гальма 1YB2';
   // DigIn_5_7.Chanal := WSTRING#'15';
   // DigIn_6_0.Text := WSTRING#'Механізм пересування візка. Термозахист гальмівного резистора';
   // DigIn_6_0.Chanal := WSTRING#'16';
   // DigIn_6_1.Text := WSTRING#'Механізм пересування візка. Дозвіл нормальної швидкості. Рух вперед';
   // DigIn_6_1.Chanal := WSTRING#'17';
   // DigIn_6_2.Text := WSTRING#'Механізм пересування візка. Дозвіл роботи. Рух вперед';
   // DigIn_6_2.Chanal := WSTRING#'18';
   // DigIn_6_3.Text := WSTRING#'Механізм пересування візка. Дозвіл нормальної швидкості. Рух назад';
   // DigIn_6_3.Chanal := WSTRING#'19';
   // DigIn_6_4.Text := WSTRING#'Механізм пересування візка. Дозвіл роботи. Рух назад';
   // DigIn_6_4.Chanal := WSTRING#'20';
   // DigIn_6_5.Text := WSTRING#'Механізм пересування візка. Дозвіл роботи (РП розєднан з приводом)';
   // DigIn_6_5.Chanal := WSTRING#'21';
   // DigIn_6_6.Text := WSTRING#'Механізм пересування візка. Температурний захист двигуна';
   // DigIn_6_6.Chanal := WSTRING#'22';
   // DigIn_6_7.Text := WSTRING#'Дозвіл роботи з будь-якої зі сторін від колони';
   // DigIn_6_7.Chanal := WSTRING#'23';
   // DigIn_7_0.Text := WSTRING#'Механізм пересування крана. Термозахист гальмівного резистора 4RT1';
   // DigIn_7_0.Chanal := WSTRING#'24';
   // DigIn_7_1.Text := WSTRING#'Механізм пересування крана. Термозахист гальмівного резистора 4RT2';
   // DigIn_7_1.Chanal := WSTRING#'25';
   // DigIn_7_2.Text := WSTRING#'Механізм пересування крана. Дозвіл нормальної швидкості. Рух вліво';
   // DigIn_7_2.Chanal := WSTRING#'26';
   // DigIn_7_3.Text := WSTRING#'Механізм пересування крана. Дозвіл нормальної швидкості. Рух управо';
   // DigIn_7_3.Chanal := WSTRING#'27';
   // DigIn_7_4.Text := WSTRING#'Механізм пересування крана. Дозвіл роботи. Рух вліво';
   // DigIn_7_4.Chanal := WSTRING#'28';
   // DigIn_7_5.Text := WSTRING#'Механізм пересування крана. Дозвіл роботи. Рух управо';
   // DigIn_7_5.Chanal := WSTRING#'29';
   // DigIn_7_6.Text := WSTRING#'Механізм пересування крана. Дозвіл роботи (РП розєднан з приводом). 4SQ41';
   // DigIn_7_6.Chanal := WSTRING#'30';
   // DigIn_7_7.Text := WSTRING#'Механізм пересування крана. Дозвіл роботи (РП розєднан з приводом). 4SQ42';
   // DigIn_7_7.Chanal := WSTRING#'31';
END_TYPE

TYPE "udtInputAnCfg"
   STRUCT
      AnIn_0 : "AnICfg";   // Контроль крутного моменту двигуна підйома
      AnIn_1 : "AnICfg";   // Резерв
      AnIn_2 : "AnICfg";   // Резерв
      AnIn_3 : "AnICfg";   // Резерв
      AnIn_4 : "AnICfg";   // Резерв
      AnIn_5 : "AnICfg";   // Резерв
      AnIn_6 : "AnICfg";   // Резерв
      AnIn_7 : "AnICfg";   // Резерв
   END_STRUCT;
   // AnIn_0.Text := WSTRING#'Контроль крутного моменту двигуна підйома';
   // AnIn_0.Chanal := WSTRING#'0';
   // AnIn_1.Text := WSTRING#'Резерв';
   // AnIn_1.Chanal := WSTRING#'1';
   // AnIn_2.Text := WSTRING#'Резерв';
   // AnIn_3.Text := WSTRING#'Резерв';
   // AnIn_4.Text := WSTRING#'Резерв';
   // AnIn_5.Text := WSTRING#'Резерв';
   // AnIn_6.Text := WSTRING#'Резерв';
   // AnIn_7.Text := WSTRING#'Резерв';
   // AnIn_2.Chanal := WSTRING#'2';
   // AnIn_3.Chanal := WSTRING#'3';
   // AnIn_4.Chanal := WSTRING#'4';
   // AnIn_5.Chanal := WSTRING#'5';
   // AnIn_6.Chanal := WSTRING#'6';
   // AnIn_7.Chanal := WSTRING#'7';
END_TYPE

TYPE "udtOutputCfg"
   STRUCT
      DigOut_0_0 : "DigOCfg";   // Включення рабочого гальма підйому
      DigOut_0_1 : "DigOCfg";   // Включення вбудованого гальма підйому
      DigOut_0_2 : "DigOCfg";   // Включення аварійного гальма підйому
      DigOut_0_3 : "DigOCfg";   // Включення рабочого гальма пересування візка
      DigOut_0_4 : "DigOCfg";   // Включення рабочих гальм пересування крана
      DigOut_0_5 : "DigOCfg";   // Дозвіл включення лінійного контактора
      DigOut_0_6 : "DigOCfg";   // Вимкнення лінійного контактора
      DigOut_0_7 : "DigOCfg";   // Включення дзвінка
      DigOut_1_0 : "DigOCfg";   // Резерв
      DigOut_1_1 : "DigOCfg";   // Резерв
      DigOut_1_2 : "DigOCfg";   // Лампа. Готовність приводу підйому
      DigOut_1_3 : "DigOCfg";   // Лампа. Готовність приводу пересування візка
      DigOut_1_4 : "DigOCfg";   // Лампа. Готовність приводу пересування крана
      DigOut_1_5 : "DigOCfg";   // Лампа. Лінійний контактор увімкнено
      DigOut_1_6 : "DigOCfg";   // Лампа. Вхідна напруга не в нормі
      DigOut_1_7 : "DigOCfg";   // Резерв
   END_STRUCT;
   // DigOut_0_0.Text := WSTRING#'Включення рабочого гальма підйому';
   // DigOut_0_0.Chanal := WSTRING#'0';
   // DigOut_0_1.Chanal := WSTRING#'1';
   // DigOut_0_2.Chanal := WSTRING#'2';
   // DigOut_0_3.Chanal := WSTRING#'3';
   // DigOut_0_4.Chanal := WSTRING#'4';
   // DigOut_0_5.Chanal := WSTRING#'5';
   // DigOut_0_6.Chanal := WSTRING#'6';
   // DigOut_0_7.Chanal := WSTRING#'7';
   // DigOut_1_0.Chanal := WSTRING#'8';
   // DigOut_1_1.Chanal := WSTRING#'9';
   // DigOut_1_2.Chanal := WSTRING#'10';
   // DigOut_1_3.Chanal := WSTRING#'11';
   // DigOut_1_4.Chanal := WSTRING#'12';
   // DigOut_1_5.Chanal := WSTRING#'13';
   // DigOut_1_6.Chanal := WSTRING#'14';
   // DigOut_1_7.Chanal := WSTRING#'15';
   // DigOut_0_1.Text := WSTRING#'Включення вбудованого гальма підйому';
   // DigOut_0_2.Text := WSTRING#'Включення аварійного гальма підйому';
   // DigOut_0_3.Text := WSTRING#'Включення рабочого гальма пересування візка';
   // DigOut_0_4.Text := WSTRING#'Включення рабочих гальм пересування крана';
   // DigOut_0_5.Text := WSTRING#'Дозвіл включення лінійного контактора';
   // DigOut_0_6.Text := WSTRING#'Вимкнення лінійного контактора';
   // DigOut_0_7.Text := WSTRING#'Включення дзвінка';
   // DigOut_1_0.Text := WSTRING#'Резерв';
   // DigOut_1_1.Text := WSTRING#'Резерв';
   // DigOut_1_2.Text := WSTRING#'Лампа. Готовність приводу підйому';
   // DigOut_1_3.Text := WSTRING#'Лампа. Готовність приводу пересування візка';
   // DigOut_1_4.Text := WSTRING#'Лампа. Готовність приводу пересування крана';
   // DigOut_1_5.Text := WSTRING#'Лампа. Лінійний контактор увімкнено';
   // DigOut_1_6.Text := WSTRING#'Лампа. Вхідна напруга не в нормі';
   // DigOut_1_7.Text := WSTRING#'Резерв';
END_TYPE

// folder: (top level)

DATA_BLOCK "Data_base"   // DB1
{ S7_Optimized_Access := 'FALSE' }
VERSION : 0.1
   VAR
      ManInterlock : "udtMDM";   // Ручне керування
      MovePerm : "udtMovePerm";   // Дозвіл роботи
      SpeedPerm : "udtSpeedPerm";   // Дозвіл ном. швидкості
      Remote_control : "udtRemCtrl";   // Пульт S1
      Ons : Array[0..99] of Bool;
      xReset : Bool;   // Скидання помилок
      Lifebit_HMI : Bool;   // Панель оператора
      Lifebit_HMI_Old : Bool;
      TestReal : Array[0..100] of Real;
      TestBool : Array[0..100] of Bool;
      Ring_Status : Int;
      ReadBytes : Int;
      RetVal : Int;
      SCALANCE_Buffer : Array[0..100] of Byte;
      Read_Buffer : Array[0..60] of Int;
      Read_Trigger : Bool;
      HMI_Online : Bool;
      Drive_Online : Bool;
      PROFINET_Status : Array[0..127] of Bool;
      Moduls_Err : Array[0..127] of Bool;
      ModulStatus : Int;
      Ring_Ok : Bool;
      Alarm_Ring_Broken_Scalance : Bool;
      Alarm_Ring_Broken_Drive : Bool;
      Alarm_Ring_Broken_HMI : Bool;
      Alarm_Station_Drive_Offline : Bool;
      Alarm_Station_HMI_Offline : Bool;
      Devices_With_Errors : Array[0..127] of Bool;
      Devices_Online : Array[0..127] of Bool;
      Devices_val_1 : Int;
      Devices_val_2 : Int;
      Devices_val_3 : Int;
      Devices_val_4 : Int;
      Devices_val_5 : Int;
      Devices_val_6 : Int;
   END_VAR
BEGIN
END_DATA_BLOCK

DATA_BLOCK "HMI_DB"   // DB10
{ S7_Optimized_Access := 'TRUE' }
VERSION : 0.1
   VAR
      IO_Tags : Struct   // Вхідні-Вихідні сигнали
         InCnf : "udtInputCfg";
         InAnCfg : "udtInputAnCfg";
         OutCfg : "udtOutputCfg";
      END_STRUCT;
      PSM : Struct   // Живлення
         Line_contactor_On : Bool;   // Лінійний контактор включений
         Control_contactor_220V_On : Bool;   // Контактор кіл управління 220В, 50Гц включений
         Input_voltage_control_380V_On : Bool;   // Контроль напруги введення, 380В, 50Гц
         Heating_circuit_breaker_220V_On : Bool;   // Вимикач кіл живлення обігріву 220В, 50Гц
         Brake_protection_On : Bool;   // Захист кіл гальм
         Transformer_6T1_380V_On : Bool;   // Вимикач трансформатора 6Т1, 380В, 50Гц
         Transformer_sec_circuit_breaker_6T1_380V_On : Bool;   // Вимикач вторинних кіл трансформатора 6Т1, 380В, 50Гц
         Power_switch_6KV_380V_On : Bool;   // Вимикач живлення 6KV, 380В, 50Гц
         ID_Control_circuit_breaker_220V_On : Bool;   // Ввідний пристрій. Вимикач кіл управління 220В, 50Гц
         ID_ORP_power_circuit_breaker_220V_On : Bool;   // Ввідний пристрій. Вимикач кіл живлення ОВП, 220В, 50Гц
         ID_Line_contactor_from_remote_control_On : Bool;   // Ввідний пристрій. Команда на включення лінійного контактора з пульта
         Transformer_9T1_380V_On : Bool;   // Вимикач трансформатора 9Т1, 380В, 50Гц
         Repair_lighting_switch_12V_On : Bool;   // Вимикач ремонтного освітлення, 12В, 50Гц
         Cabinet_circuit_breaker_220V_On : Bool;   // Вимикач власних потреб шафа, 220В, 50Гц
         CMD_Line_contactor_enable_permission : Bool;   // Дозвіл включення лінійного контактора
         CMD_Line_contactor_Off : Bool;   // Вимкнення лінійного контактора
         HL_Line_contactor_On : Bool;   // Лампа. Лінійний контактор увімкнено
         HL_Input_voltage_abnormal : Bool;   // Лампа. Вхідна напруга не в нормі
         Zero_Protection : Bool;   // Активовано блокування «Нульовий захист»
         LC_Alarm : Bool;   // Загальний прапор критичної аварії контактора
         ColumnEnable : Bool;   // Дозвіл переміщення за колоною
         AlarmWord : Word;   // Код помилки лінейного контактора для панелі ЛМІ
         TripWord_1 : Word;   // Код причини аварійного відключення контактора
         TripWord_2 : Word;   // Код причини аварійного відключення контактора
      END_STRUCT;
      Sensors : Struct   // Сенсори
         Cabinet_heating_control_SU1 : Bool;   // Контроль підігріву шафи SU1
         Seismic_sensor : Bool;   // Сейсмодатчик
         Drum_rotation_control : Bool;   // Контроль обертання барабану
         CMD_Bell_On : Bool;   // Включення дзвінка
      END_STRUCT;
      Encoders : Struct   // Екодери
         "1BR" : "UDT_HMI_Encoder_View";   // Енкодер підйома
         "3BR" : "UDT_HMI_Encoder_View";   // Енкодер пересування візка
         "4BR1" : "UDT_HMI_Encoder_View";   // Енкодер#1 пересування крана
         "4BR2" : "UDT_HMI_Encoder_View";   // Енкодер#2 пересування крана
      END_STRUCT;
      Remote_control : "udtRemCtrl";   // Пульт S1
      Drives : Struct   // Приводи
         CU_U1 : "UDT_HMI_S120_CU";   // Блок управління приводами U1 CU320-2 PN
         Drive_1UZ1 : "UDT_HMI_S120_Drive";   // ПЧ 1UZ1
         Drive_3UZ1 : "UDT_HMI_S120_Drive";   // ПЧ 3UZ1
         Drive_4UZ1 : "UDT_HMI_S120_Drive";   // ПЧ 4UZ1
         Drive_4UZ2 : "UDT_HMI_S120_Drive";   // ПЧ 4UZ2
      END_STRUCT;
      Lifting_mechanism : Struct   // Механізм підйому (Hoist) / Механізм підйому
         Work_control : Bool;   // Контроль роботи механізму підйому
         Brake_wear_control : Bool;   // Контроль зносу гальма механізму підйому
         MD_disconnected_from_drive : Bool;   // Механізм підйому. РП роз'єднаний з приводом
         Thermal_protection_braking_resistor : Bool;   // Механізм підйому. Термозахист гальмівного резистора
         NSP_Upward_movement : Bool;   // Механізм підйому. Дозвіл нормальної швидкості. Рух вгору
         NSP_Downward_movement : Bool;   // Механізм підйому. Дозвіл нормальної швидкості. Рух вниз
         WP_Upward_movement : Bool;   // Механізм підйому. Дозвіл роботи. Рух вгору
         WP_Downward_movement : Bool;   // Механізм підйому. Дозвіл роботи. Рух вниз
         "Exceeding_rated_load_115%" : Bool;   // Механізм підйому. Перевищення номінального вантажу 115%
         Loosening_ropes : Bool;   // Механізм підйому. Ослаблення канатів
         Motor_temperature_protection : Bool;   // Механізм підйому. Температурний захист двигуна
         "1YB1_Brake released" : Bool;   // Механізм підйому. Вимикачі кінцеві на гальмі 1YB1. Гальмо розгальмоване
         "1YB1_Brake_applied" : Bool;   // Механізм підйому. Вимикачі кінцеві на гальмі 1YB1. Гальмо загальмоване
         "1YB1_Thickness_brake_pads_normal" : Bool;   // Механізм підйому. Вимикачі кінцеві на гальмі 1YB1. Товщина гальмівних наладок в нормі
         "1YB2_Brake released" : Bool;   // Механізм підйому. Вимикачі кінцеві на гальмі 1YB2. Гальмо розгальмоване
         "1YB2_Brake_applied" : Bool;   // Механізм підйому. Вимикачі кінцеві на гальмі 1YB2. Гальмо загальмоване
         "1YB2_WP_MPP_disconnected_from_brake" : Bool;   // Механізм підйому. Вимикачі кінцеві на гальмі 1YB2. Дозвіл роботи (MPP роз'єднаний з гальмом)
         "1YB1_Brake_rectifier_protection" : Bool;   // Механізм підйому. Захист випрямляча гальма 1YB1
         "1YB2_Brake_rectifier_protection" : Bool;   // Механізм підйому. Захист випрямляча гальма 1YB2
         CMD_Service_brake_On : Bool;   // Включення рабочого гальма підйому
         "CMD_Built-in_brake_On" : Bool;   // Включення вбудованого гальма підйому
         CMD_Emergency_brake_On : Bool;   // Включення аварійного гальма підйому
         HL_Drive_ready : Bool;   // Лампа. Готовність приводу підйому
         Torque_control : Real;   // Контроль крутного моменту двигуна підйома
         LM_Alarm : Bool;   // Загальний прапор критичної аварії механізма підйому
         NSP_Enable_movement : Bool;   // Загальний сигнал дозволу номінальної швидкості
         SecondSpeedUp : Bool;   // Команда 2-га швидкість Вверх
         SecondSpeedDown : Bool;   // Команда 2-га швидкість Вниз
         FirstSpeedUp : Bool;   // Команда 1-ша швидкість Вверх
         FirstSpeedDown : Bool;   // Команда 1-ша швидкість Вниз
         LM_Status : Word;   // Слово стану підйомника
      END_STRUCT;
      Trolley_movement_mechanism : Struct   // Механізм пересування візка
         Engine_temperature_protection : Bool;   // Механізм пересування візка. Термозахист гальмівного резистора
         NSP_Forward_movement : Bool;   // Механізм пересування візка. Дозвіл нормальної швидкості. Рух вперед
         WP_Forward_movement : Bool;   // Механізм пересування візка. Дозвіл роботи. Рух вперед
         NSP_Backward_movement : Bool;   // Механізм пересування візка. Дозвіл нормальної швидкості. Рух назад
         WP_Backward_movement : Bool;   // Механізм пересування візка. Дозвіл роботи. Рух назад
         MD_disconnected_from_drive : Bool;   // Механізм пересування візка. Дозвіл роботи (РП роз'єднан з приводом)
         Motor_temperature_protection : Bool;   // Механізм пересування візка. Температурний захист двигуна
         CMD_Service_brake_On : Bool;   // Включення рабочого гальма пересування візка
         HL_Drive_ready : Bool;   // Лампа. Готовність приводу пересування візка
         TM_Alarm : Bool;   // Загальний прапор критичної аварії механізма підйому / Загальний прапор критичної аварії механізма переміщення візка
         NSP_Enable_movement : Bool;   // Загальний сигнал дозволу номінальної швидкості
         SecondSpeedForward : Bool;   // Команда 2-га швидкість Вперед
         SecondSpeedBackward : Bool;   // Команда 2-га швидкість Назад
         FirstSpeedForward : Bool;   // Команда 1-ша швидкість Вперед
         FirstSpeedBackward : Bool;   // Команда 1-ша швидкість Назад
         TM_Status : Word;   // Слово стану візка
      END_STRUCT;
      Crane_movement_mechanism : Struct   // Механізм пересування крана
         Brake_protection_On : Bool;   // Механізм пересування крана. Захист кіл гальм
         "4M1_engine_temperature_protection" : Bool;   // Механізм пересування крана. Температурний захист двигуна 4M1
         "4M2_engine_temperature_protection" : Bool;   // Механізм пересування крана. Температурний захист двигуна 4M2
         WP_Either_side_column : Bool;   // Механізм пересування крана. Дозвіл роботи з будь-якої зі сторін від колони
         "4RT1_thermal_protection_braking_resistor" : Bool;   // Механізм пересування крана. Термозахист гальмівного резистора 4RT1
         "4RT2_thermal_protection_braking_resistor" : Bool;   // Механізм пересування крана. Термозахист гальмівного резистора 4RT2
         NSP_Left_movement : Bool;   // Механізм пересування крана. Дозвіл нормальної швидкості. Рух вліво
         NSP_Right_movement : Bool;   // Механізм пересування крана. Дозвіл нормальної швидкості. Рух управо
         WP_Left_movement : Bool;   // Механізм пересування крана. Дозвіл роботи. Рух вліво
         WP_Right_movement : Bool;   // Механізм пересування крана. Дозвіл роботи. Рух управо
         "4SQ41_MD_disconnected_from_drive" : Bool;   // Механізм пересування крана. Дозвіл роботи (РП роз'єднан з приводом). 4SQ41
         "4SQ42_MD_disconnected_from_drive" : Bool;   // Механізм пересування крана. Дозвіл роботи (РП роз'єднан з приводом). 4SQ42
         CMD_Service_brake_On : Bool;   // Включення рабочих гальм пересування крана
         HL_Drive_ready : Bool;   // Лампа. Готовність приводу пересування крана
         NSP_Enable_movement : Bool;   // Загальний сигнал дозволу номінальної швидкості
         BreakThermalProtection : Bool;   // Загальний сигнал термозахисту гальмівних резисторів
         MotorThermalProtection : Bool;   // Загальний сигнал термозахист двигунів
         SecondSpeedLeft : Bool;   // Команда 2-га швидкість Вліво
         SecondSpeedRight : Bool;   // Команда 2-га швидкість Вправо
         FirstSpeedLeft : Bool;   // Команда 1-ша швидкість Вліво
         FirstSpeedRight : Bool;   // Команда 1-ша швидкість Вправо
         Max_Skew_Limit : DInt := 50;   // Максимальна межа перекосу
         CM_Status : Word;   // Слово стану крана
         CM_Alarm : Bool;   // Загальний прапор критичної аварії механізма підйому / Загальний прапор критичної аварії механізма переміщення крана
      END_STRUCT;
      Reserv : Struct   // Резерв
         I3_0 : Bool;
         Q1_0 : Bool;
         Q1_1 : Bool;
         Q1_7 : Bool;
         IW10 : Real;
         IW12 : Real;
         IW14 : Real;
         IW16 : Real;
         IW18 : Real;
         IW20 : Real;
         IW22 : Real;
      END_STRUCT;
      Messages : Struct   // Сповіщення
         LinearContactor : Struct
            wMessageWord1 : Word;
            wMessageWord2 : Word;
            wMessageWord3 : Word;
            wMessageWord4 : Word;
            wMessageWord5 : Word;
         END_STRUCT;
         LiftUp : Struct
            wMessageWord1 : Word;
            wMessageWord2 : Word;
            wMessageWord3 : Word;
            wMessageWord4 : Word;
         END_STRUCT;
         Trolley : Struct
            wMessageWord1 : Word;
            wMessageWord2 : Word;
            wMessageWord3 : Word;
         END_STRUCT;
         Crane : Struct
            wMessageWord1 : Word;
            wMessageWord2 : Word;
            wMessageWord3 : Word;
         END_STRUCT;
         Diag : Struct
            wMessageWord1 : Word;
            wMessageWord2 : Word;
         END_STRUCT;
         Self : Struct
            wMessageWord1 : Word;
         END_STRUCT;
      END_STRUCT;
      Alarms : Struct   // Аварії
         Contactor : Struct
            AlarmWord1 : Word;
            AlarmWord2 : Word;
            AlarmWord3 : Word;
         END_STRUCT;
         LiftUp : Struct
            AlarmWord1 : Word;
            AlarmWord2 : Word;
         END_STRUCT;
         Trolley : Struct
            AlarmWord1 : Word;
            AlarmWord2 : Word;
         END_STRUCT;
         Crane : Struct
            AlarmWord1 : Word;
            AlarmWord2 : Word;
         END_STRUCT;
         Diagnose : Struct
            AlarmWord1 : Word;
         END_STRUCT;
      END_STRUCT;
      Warnings : Struct   // Попередження
         LiftUp : Word;
         Trolley : Word;
         Crane : Word;
      END_STRUCT;
      Diagnostics : Struct   // Діагностика
         PLC_Ok : Bool;
         SCALANCE_Ok : Bool;
         "1BR_Ok" : Bool;
         "3BR_Ok" : Bool;
         "4BK1_Ok" : Bool;
         "4BR2_Ok" : Bool;
         CU320_Ok : Bool;
         Profinet_Ok : Bool;
         HMI_Flt : Bool;
         PLC_Flt : Bool;
         A1_2_LED_Status : Int;
         A1_3_LED_Status : Int;
         A1_4_LED_Status : Int;
         A1_5_LED_Status : Int;
         "A1.2_Flt" : Bool;
         "A1.3_Flt" : Bool;
         "A1.4_Flt" : Bool;
         "A1.5_Flt" : Bool;
         "A1.6_Flt" : Bool;
         "1BR_Flt" : Bool;
         "3BR_Flt" : Bool;
         "4BR1_Flt" : Bool;
         "4BR2_Flt" : Bool;
         U1_Flt : Bool;
         "1UZ1_Flt" : Bool;
         "3UZ1_Flt" : Bool;
         "4UZ1_Flt" : Bool;
         "4UZ2_Flt" : Bool;
         Ring_PLC_HMI_NOK : Bool;   // Порушено кільце між ПЛК та ЛМІ
         Ring_PLC_SCALAMCE_NOK : Bool;   // Порушено кільце між ПЛК та Світчем
         Ring_HMI_CU_NOK : Bool;   // Порушено кільце між ЛМІ та ПЧ
         Ring_SCALAMCE_CU_NOK : Bool;   // Порушено кільце між Світчем та ПЧ
      END_STRUCT;
      wCoordination : Word;   // Coordination signal
      wButtonHighlight : Word;
      Calibration : Struct   // Калібровка
         Hoist : Struct   // Підйом
            Active : Bool := FALSE;   // Процедура калібровки підйому активна
            Calibrated : Bool := FALSE;   // Механізм підйому відкалібровано
            Fault : Bool := FALSE;   // Помилка процедури калібровки
            Aborted : Bool := FALSE;   // Процедуру калібровки перервано
            CurrentStep : UInt := UINT#0;   // Поточний крок калібровки
            CompletedSteps : DWord := DWORD#0;   // Бітова маска завершених кроків калібровки
            Reference1K1 : Bool := FALSE;   // Поточний стан реперного кінцевика 1K1
            Position_mm : DInt := 0;   // Поточне положення механізму підйому, мм
            DriveVelocity_rpm : Real := 0.0;   // Фактична швидкість привода, об/хв
            TimerRemaining : Time := T#0ms;   // Залишок часу активного таймера
            TimerRemaining_Min : UInt;   // Залишок повних хвилин часу активного таймера
            TimerRemaining_Sec : UInt;   // Залишок секунд часу активного таймера
            Steps_Completed : Struct   // Завершені кроки
               Step10 : Bool;   // Крок 10 «Перевірка умов» виконано
               Step20 : Bool;   // Крок 20 «Команда Підйом» виконано
               Step30 : Bool;   // Крок 30 «Перший підхід до 1K1» виконано
               Step40 : Bool;   // Крок 40 «Відпускання кнопки Підйом» виконано
               Step50 : Bool;   // Крок 50 «Відхід вниз» виконано
               Step60 : Bool;   // Крок 60 «Відхід завершено» виконано
               Step70 : Bool;   // Крок 70 «Повторна команда Підйом» виконано
               Step80 : Bool;   // Крок 80 «Повторний підхід до 1K1» виконано
               Step90 : Bool;   // Крок 90 «Quick Stop» виконано
               Step100 : Bool;   // Крок 100 «Привід зупинено» виконано
               Step110 : Bool;   // Крок 110 «Preset запущено» виконано
               Step120 : Bool;   // Крок 120 «Preset завершено» виконано
               Step130 : Bool;   // Крок 130 «Калібровка завершена» виконано
            END_STRUCT;
            Steps_Active : Struct   // Активні кроки
               Step10 : Bool;   // Крок 10 «Перевірка умов» активний
               Step20 : Bool;   // Крок 20 «Команда Підйом» активний
               Step30 : Bool;   // Крок 30 «Перший підхід до 1K1» активний
               Step40 : Bool;   // Крок 40 «Відпускання кнопки Підйом» активний
               Step50 : Bool;   // Крок 50 «Відхід вниз» активний
               Step60 : Bool;   // Крок 60 «Відхід завершено» активний
               Step70 : Bool;   // Крок 70 «Повторна команда Підйом» активний
               Step80 : Bool;   // Крок 80 «Повторний підхід до 1K1» активний
               Step90 : Bool;   // Крок 90 «Quick Stop» активний
               Step100 : Bool;   // Крок 100 «Привід зупинено» активний
               Step110 : Bool;   // Крок 110 «Preset запущено» активний
               Step120 : Bool;   // Крок 120 «Preset завершено» активний
               Step130 : Bool;   // Крок 130 «Калібровка завершена» активний
            END_STRUCT;
            Diagnostics : Struct   // Діагностика
               EncoderControlHealthy : Bool := FALSE;   // Справність контролю енкодера
               StartupDataConsistent : Bool := TRUE;   // Дані енкодера після увімкнення PLC узгоджені
               NoMovementWithoutCommand : Bool := TRUE;   // Не виявлено зміни положення без команди руху
               NoManualMovementDetected : Bool := TRUE;   // Не виявлено нештатного переміщення без активації ручного приводу
               EncoderUpdatesDuringMotion : Bool := TRUE;   // Значення енкодера оновлюються під час руху
               EncoderReplacementNotDetected : Bool := TRUE;   // Фізичну заміну енкодера не виявлено
            END_STRUCT;
         END_STRUCT;
         Trolley : Struct   // Візок
            Active : Bool := FALSE;   // Процедура калібровки візка активна
            Calibrated : Bool := FALSE;   // Механізм візка відкалібровано
            Fault : Bool := FALSE;   // Помилка процедури калібровки
            Aborted : Bool := FALSE;   // Процедуру калібровки перервано
            PrerequisitesNotOK : Bool := FALSE;   // Не виконані початкові умови калібровки візка
            CurrentStep : UInt := UINT#0;   // Поточний крок калібровки
            CompletedSteps : DWord := DWORD#0;   // Бітова маска завершених кроків
            Reference3K1 : Bool := FALSE;   // Поточний стан реперного вимикача 3K1
            Position_mm : DInt := 0;   // Поточне положення візка, мм
            DriveVelocity_rpm : Real := 0.0;   // Фактична швидкість привода візка, об/хв
            TimerRemaining : Time := T#0ms;   // Залишок часу активного таймера
            TimerRemaining_Min : UInt := 0;   // Залишок повних хвилин
            TimerRemaining_Sec : UInt := 0;   // Залишок секунд
            Steps_Completed : Struct   // Завершені кроки
               Step10 : Bool := FALSE;   // Крок 10 «Перевірка умов» виконано
               Step20 : Bool := FALSE;   // Крок 20 «Команда Вперед» виконано
               Step30 : Bool := FALSE;   // Крок 30 «Перший підхід до 3K1» виконано
               Step40 : Bool := FALSE;   // Крок 40 «Відпускання кнопки Вперед» виконано
               Step50 : Bool := FALSE;   // Крок 50 «Відхід назад» виконано
               Step60 : Bool := FALSE;   // Крок 60 «Відхід завершено» виконано
               Step70 : Bool := FALSE;   // Крок 70 «Повторна команда Вперед» виконано
               Step80 : Bool := FALSE;   // Крок 80 «Повторний підхід до 3K1» виконано
               Step90 : Bool := FALSE;   // Крок 90 «Quick Stop» виконано
               Step100 : Bool := FALSE;   // Крок 100 «Привід зупинено» виконано
               Step110 : Bool := FALSE;   // Крок 110 «Preset запущено» виконано
               Step120 : Bool := FALSE;   // Крок 120 «Preset завершено» виконано
               Step130 : Bool := FALSE;   // Крок 130 «Калібровка завершена» виконано
            END_STRUCT;
            Steps_Active : Struct   // Активні кроки
               Step10 : Bool := FALSE;   // Крок 10 «Перевірка умов» активний
               Step20 : Bool := FALSE;   // Крок 20 «Команда Вперед» активний
               Step30 : Bool := FALSE;   // Крок 30 «Перший підхід до 3K1» активний
               Step40 : Bool := FALSE;   // Крок 40 «Відпускання кнопки Вперед» активний
               Step50 : Bool := FALSE;   // Крок 50 «Відхід назад» активний
               Step60 : Bool := FALSE;   // Крок 60 «Відхід завершено» активний
               Step70 : Bool := FALSE;   // Крок 70 «Повторна команда Вперед» активний
               Step80 : Bool := FALSE;   // Крок 80 «Повторний підхід до 3K1» активний
               Step90 : Bool := FALSE;   // Крок 90 «Quick Stop» активний
               Step100 : Bool := FALSE;   // Крок 100 «Привід зупинено» активний
               Step110 : Bool := FALSE;   // Крок 110 «Preset запущено» активний
               Step120 : Bool := FALSE;   // Крок 120 «Preset завершено» активний
               Step130 : Bool := FALSE;   // Крок 130 «Калібровка завершена» активний
            END_STRUCT;
            Diagnostics : Struct   // Діагностика
               EncoderControlHealthy : Bool := FALSE;   // Справність контролю енкодера 3BR
               StartupDataConsistent : Bool := TRUE;   // Дані енкодера після увімкнення PLC узгоджені
               NoMovementWithoutCommand : Bool := TRUE;   // Не виявлено зміни положення без команди руху
               NoManualMovementDetected : Bool := TRUE;   // Не виявлено нештатного переміщення без ручного приводу
               EncoderUpdatesDuringMotion : Bool := TRUE;   // Значення енкодера оновлюються під час руху
               EncoderReplacementNotDetected : Bool := TRUE;   // Фізичну заміну енкодера не виявлено
            END_STRUCT;
         END_STRUCT;
         Crane : Struct   // Міст
            Active : Bool := FALSE;   // Процедура калібровки моста активна
            Calibrated : Bool := FALSE;   // Механізм моста відкалібровано
            Fault : Bool := FALSE;   // Помилка процедури калібровки
            Aborted : Bool := FALSE;   // Процедуру калібровки перервано
            PrerequisitesNotOK : Bool := FALSE;   // Не виконані початкові умови калібровки моста
            CurrentStep : UInt := UINT#0;   // Поточний крок калібровки
            CompletedSteps : DWord := DWORD#0;   // Бітова маска завершених кроків калібровки
            Reference4K1 : Bool := FALSE;   // Поточний стан реперного вимикача 4K1
            Position4BR1_mm : DInt := 0;   // Поточна позиція моста за енкодером 4BR1, мм
            Position4BR2_mm : DInt := 0;   // Поточна позиція моста за енкодером 4BR2, мм
            Drive1Velocity_rpm : Real := 0.0;   // Фактична швидкість привода 4UZ1, об/хв
            Drive2Velocity_rpm : Real := 0.0;   // Фактична швидкість привода 4UZ2, об/хв
            TimerRemaining : Time := T#0ms;   // Залишок часу активного таймера
            TimerRemaining_Min : UInt := 0;   // Залишок повних хвилин
            TimerRemaining_Sec : UInt := 0;   // Залишок секунд
            Steps_Completed : Struct   // Завершені кроки
               Step10 : Bool;   // Крок 10 «Перевірка умов» виконано
               Step20 : Bool;   // Крок 20 «Команда Вліво» виконано
               Step30 : Bool;   // Крок 30 «Перший підхід до 4K1» виконано
               Step40 : Bool;   // Крок 40 «Відпускання кнопки Вліво» виконано
               Step50 : Bool;   // Крок 50 «Відхід вправо» виконано
               Step60 : Bool;   // Крок 60 «Відхід завершено» виконано
               Step70 : Bool;   // Крок 70 «Повторна команда Вліво» виконано
               Step80 : Bool;   // Крок 80 «Повторний підхід до 4K1» виконано
               Step90 : Bool;   // Крок 90 «Quick Stop» виконано
               Step100 : Bool;   // Крок 100 «Приводи зупинено» виконано
               Step110 : Bool;   // Крок 110 «Preset запущено» виконано
               Step120 : Bool;   // Крок 120 «Preset завершено» виконано
               Step130 : Bool;   // Крок 130 «Калібровка завершена» виконано
            END_STRUCT;
            Steps_Active : Struct   // Активні кроки
               Step10 : Bool;   // Крок 10 «Перевірка умов» активний
               Step20 : Bool;   // Крок 20 «Команда Вліво» активний
               Step30 : Bool;   // Крок 30 «Перший підхід до 4K1» активний
               Step40 : Bool;   // Крок 40 «Відпускання кнопки Вліво» активний
               Step50 : Bool;   // Крок 50 «Відхід вправо» активний
               Step60 : Bool;   // Крок 60 «Відхід завершено» активний
               Step70 : Bool;   // Крок 70 «Повторна команда Вліво» активний
               Step80 : Bool;   // Крок 80 «Повторний підхід до 4K1» активний
               Step90 : Bool;   // Крок 90 «Quick Stop» активний
               Step100 : Bool;   // Крок 100 «Приводи зупинено» активний
               Step110 : Bool;   // Крок 110 «Preset запущено» активний
               Step120 : Bool;   // Крок 120 «Preset завершено» активний
               Step130 : Bool;   // Крок 130 «Калібровка завершена» активний
            END_STRUCT;
            Diagnostics : Struct   // Діагностика
               Encoder1ControlHealthy : Bool := FALSE;   // Справність контролю енкодера 4BR1
               Encoder1StartupDataConsistent : Bool := TRUE;   // Дані 4BR1 після увімкнення PLC узгоджені
               Encoder1NoMovementWithoutCommand : Bool := TRUE;   // Не виявлено зміни положення 4BR1 без команди руху
               Encoder1NoManualMovementDetected : Bool := TRUE;   // Не виявлено нештатного переміщення 4BR1 без ручного приводу
               Encoder1UpdatesDuringMotion : Bool := TRUE;   // Значення 4BR1 оновлюються під час руху
               Encoder1ReplacementNotDetected : Bool := TRUE;   // Фізичну заміну 4BR1 не виявлено
               Encoder2ControlHealthy : Bool := FALSE;   // Справність контролю енкодера 4BR2
               Encoder2StartupDataConsistent : Bool := TRUE;   // Дані 4BR2 після увімкнення PLC узгоджені
               Encoder2NoMovementWithoutCommand : Bool := TRUE;   // Не виявлено зміни положення 4BR2 без команди руху
               Encoder2NoManualMovementDetected : Bool := TRUE;   // Не виявлено нештатного переміщення 4BR2 без ручного приводу
               Encoder2UpdatesDuringMotion : Bool := TRUE;   // Значення 4BR2 оновлюються під час руху
               Encoder2ReplacementNotDetected : Bool := TRUE;   // Фізичну заміну 4BR2 не виявлено
               EncoderDifferenceOK : Bool := TRUE;   // Розбіжність показань 4BR1 та 4BR2 не перевищує допустиму
               DiagnosticsHealthy : Bool := FALSE;   // Усі реалізовані контролі діагностики моста в нормі
               DriveStandstill : Bool := FALSE;   // Обидва приводи моста повністю зупинені
               EncoderDifference_mm : LReal := 0.0;   // Поточна розбіжність між 4BR1 та 4BR2, мм
               Position1DeltaStopped_mm : LReal := 0.0;   // Зміна позиції 4BR1 від точки зупинки
               Position2DeltaStopped_mm : LReal := 0.0;   // Зміна позиції 4BR2 від точки зупинки
               Position1DeltaMotion_mm : LReal := 0.0;   // Зміна позиції 4BR1 для watchdog руху
               Position2DeltaMotion_mm : LReal := 0.0;   // Зміна позиції 4BR2 для watchdog руху
            END_STRUCT;
         END_STRUCT;
      END_STRUCT;
      FireAlarm : Struct   // Пожежна сигналізація
         Active : Bool;   // Пожежна сигналізація активна
      END_STRUCT;
   END_VAR
BEGIN
   IO_Tags.InCnf.DigIn_0_0.Chanal := WSTRING#'I0.0';
   IO_Tags.InCnf.DigIn_0_1.Chanal := WSTRING#'I0.1';
   IO_Tags.InCnf.DigIn_0_2.Chanal := WSTRING#'I0.2';
   IO_Tags.InCnf.DigIn_0_3.Chanal := WSTRING#'I0.3';
   IO_Tags.InCnf.DigIn_0_4.Chanal := WSTRING#'I0.4';
   IO_Tags.InCnf.DigIn_0_5.Chanal := WSTRING#'I0.5';
   IO_Tags.InCnf.DigIn_0_6.Chanal := WSTRING#'I0.6';
   IO_Tags.InCnf.DigIn_0_7.Chanal := WSTRING#'I0.7';
   IO_Tags.InCnf.DigIn_1_0.Chanal := WSTRING#'I1.0';
   IO_Tags.InCnf.DigIn_1_1.Chanal := WSTRING#'I1.1';
   IO_Tags.InCnf.DigIn_1_2.Chanal := WSTRING#'I1.2';
   IO_Tags.InCnf.DigIn_1_3.Chanal := WSTRING#'I1.3';
   IO_Tags.InCnf.DigIn_1_4.Chanal := WSTRING#'I1.4';
   IO_Tags.InCnf.DigIn_1_5.Chanal := WSTRING#'I1.5';
   IO_Tags.InCnf.DigIn_1_6.Chanal := WSTRING#'I1.6';
   IO_Tags.InCnf.DigIn_1_7.Chanal := WSTRING#'I1.7';
   IO_Tags.InCnf.DigIn_2_0.Chanal := WSTRING#'I2.0';
   IO_Tags.InCnf.DigIn_2_1.Chanal := WSTRING#'I2.1';
   IO_Tags.InCnf.DigIn_2_2.Chanal := WSTRING#'I2.2';
   IO_Tags.InCnf.DigIn_2_3.Chanal := WSTRING#'I2.3';
   IO_Tags.InCnf.DigIn_2_4.Chanal := WSTRING#'I2.4';
   IO_Tags.InCnf.DigIn_2_5.Chanal := WSTRING#'I2.5';
   IO_Tags.InCnf.DigIn_2_6.Chanal := WSTRING#'I2.6';
   IO_Tags.InCnf.DigIn_2_7.Chanal := WSTRING#'I2.7';
   IO_Tags.InCnf.DigIn_3_0.Chanal := WSTRING#'I3.0';
   IO_Tags.InCnf.DigIn_3_1.Chanal := WSTRING#'I3.1';
   IO_Tags.InCnf.DigIn_3_2.Chanal := WSTRING#'I3.2';
   IO_Tags.InCnf.DigIn_3_3.Chanal := WSTRING#'I3.3';
   IO_Tags.InCnf.DigIn_3_4.Chanal := WSTRING#'I3.4';
   IO_Tags.InCnf.DigIn_3_5.Chanal := WSTRING#'I3.5';
   IO_Tags.InCnf.DigIn_3_6.Chanal := WSTRING#'I3.6';
   IO_Tags.InCnf.DigIn_3_7.Chanal := WSTRING#'I3.7';
   IO_Tags.InCnf.DigIn_4_0.Chanal := WSTRING#'I4.0';
   IO_Tags.InCnf.DigIn_4_1.Chanal := WSTRING#'I4.1';
   IO_Tags.InCnf.DigIn_4_2.Chanal := WSTRING#'I4.2';
   IO_Tags.InCnf.DigIn_4_3.Chanal := WSTRING#'I4.3';
   IO_Tags.InCnf.DigIn_4_4.Chanal := WSTRING#'I4.4';
   IO_Tags.InCnf.DigIn_4_5.Chanal := WSTRING#'I4.5';
   IO_Tags.InCnf.DigIn_4_6.Chanal := WSTRING#'I4.6';
   IO_Tags.InCnf.DigIn_4_7.Chanal := WSTRING#'I4.7';
   IO_Tags.InCnf.DigIn_5_0.Chanal := WSTRING#'I5.0';
   IO_Tags.InCnf.DigIn_5_1.Chanal := WSTRING#'I5.1';
   IO_Tags.InCnf.DigIn_5_2.Chanal := WSTRING#'I5.2';
   IO_Tags.InCnf.DigIn_5_3.Chanal := WSTRING#'I5.3';
   IO_Tags.InCnf.DigIn_5_4.Chanal := WSTRING#'I5.4';
   IO_Tags.InCnf.DigIn_5_5.Chanal := WSTRING#'I5.5';
   IO_Tags.InCnf.DigIn_5_6.Chanal := WSTRING#'I5.6';
   IO_Tags.InCnf.DigIn_5_7.Chanal := WSTRING#'I5.7';
   IO_Tags.InCnf.DigIn_6_0.Chanal := WSTRING#'I6.0';
   IO_Tags.InCnf.DigIn_6_1.Chanal := WSTRING#'I6.1';
   IO_Tags.InCnf.DigIn_6_2.Chanal := WSTRING#'I6.2';
   IO_Tags.InCnf.DigIn_6_3.Chanal := WSTRING#'I6.3';
   IO_Tags.InCnf.DigIn_6_4.Chanal := WSTRING#'I6.4';
   IO_Tags.InCnf.DigIn_6_5.Chanal := WSTRING#'I6.5';
   IO_Tags.InCnf.DigIn_6_6.Chanal := WSTRING#'I6.6';
   IO_Tags.InCnf.DigIn_6_7.Chanal := WSTRING#'I6.7';
   IO_Tags.InCnf.DigIn_7_0.Chanal := WSTRING#'I7.0';
   IO_Tags.InCnf.DigIn_7_1.Chanal := WSTRING#'I7.1';
   IO_Tags.InCnf.DigIn_7_2.Chanal := WSTRING#'I7.2';
   IO_Tags.InCnf.DigIn_7_3.Chanal := WSTRING#'I7.3';
   IO_Tags.InCnf.DigIn_7_4.Chanal := WSTRING#'I7.4';
   IO_Tags.InCnf.DigIn_7_5.Chanal := WSTRING#'I7.5';
   IO_Tags.InCnf.DigIn_7_6.Chanal := WSTRING#'I7.6';
   IO_Tags.InCnf.DigIn_7_7.Chanal := WSTRING#'I7.7';
   IO_Tags.InAnCfg.AnIn_0.Chanal := WSTRING#'IW8';
   IO_Tags.InAnCfg.AnIn_1.Chanal := WSTRING#'IW10';
   IO_Tags.InAnCfg.AnIn_2.Chanal := WSTRING#'IW12';
   IO_Tags.InAnCfg.AnIn_3.Chanal := WSTRING#'IW14';
   IO_Tags.InAnCfg.AnIn_4.Chanal := WSTRING#'IW16';
   IO_Tags.InAnCfg.AnIn_5.Chanal := WSTRING#'IW18';
   IO_Tags.InAnCfg.AnIn_6.Chanal := WSTRING#'IW20';
   IO_Tags.InAnCfg.AnIn_7.Chanal := WSTRING#'IW22';
   IO_Tags.OutCfg.DigOut_0_0.Chanal := WSTRING#'Q0.0';
   IO_Tags.OutCfg.DigOut_0_1.Chanal := WSTRING#'Q0.1';
   IO_Tags.OutCfg.DigOut_0_2.Chanal := WSTRING#'Q0.2';
   IO_Tags.OutCfg.DigOut_0_3.Chanal := WSTRING#'Q0.3';
   IO_Tags.OutCfg.DigOut_0_4.Chanal := WSTRING#'Q0.4';
   IO_Tags.OutCfg.DigOut_0_5.Chanal := WSTRING#'Q0.5';
   IO_Tags.OutCfg.DigOut_0_6.Chanal := WSTRING#'Q0.6';
   IO_Tags.OutCfg.DigOut_0_7.Chanal := WSTRING#'Q0.7';
   IO_Tags.OutCfg.DigOut_1_0.Chanal := WSTRING#'Q1.0';
   IO_Tags.OutCfg.DigOut_1_1.Chanal := WSTRING#'Q1.1';
   IO_Tags.OutCfg.DigOut_1_2.Chanal := WSTRING#'Q1.2';
   IO_Tags.OutCfg.DigOut_1_3.Chanal := WSTRING#'Q1.3';
   IO_Tags.OutCfg.DigOut_1_4.Chanal := WSTRING#'Q1.4';
   IO_Tags.OutCfg.DigOut_1_5.Chanal := WSTRING#'Q1.5';
   IO_Tags.OutCfg.DigOut_1_6.Chanal := WSTRING#'Q1.6';
   IO_Tags.OutCfg.DigOut_1_7.Chanal := WSTRING#'Q1.7';
   IO_Tags.InCnf.DigIn_5_5.Text := WSTRING#'Підйом: КВ гальма 1YB2, дозв. МРР';
   IO_Tags.InCnf.DigIn_5_2.Text := WSTRING#'Підйом: КВ накладок гальма 1YB1';
   IO_Tags.InCnf.DigIn_0_0.Text := WSTRING#'Лін. контактор увімкн.';
   IO_Tags.InCnf.DigIn_0_1.Text := WSTRING#'Контактор кіл керування 220 В увімкн.';
   IO_Tags.InCnf.DigIn_0_2.Text := WSTRING#'Контроль ввідної напруги 380 В';
   IO_Tags.InCnf.DigIn_0_3.Text := WSTRING#'Автомат обігріву 220 В';
   IO_Tags.InCnf.DigIn_0_4.Text := WSTRING#'Захист кіл гальм';
   IO_Tags.InCnf.DigIn_0_5.Text := WSTRING#'Автомат трансформатора 6T1';
   IO_Tags.InCnf.DigIn_0_6.Text := WSTRING#'Автомат втор. кіл 6T1';
   IO_Tags.InCnf.DigIn_0_7.Text := WSTRING#'Автомат реле контролю напруги';
   IO_Tags.InCnf.DigIn_1_0.Text := WSTRING#'Ввідний пристрій: автомат кіл керування';
   IO_Tags.InCnf.DigIn_1_1.Text := WSTRING#'Ввідний пристрій: автомат кіл живлення';
   IO_Tags.InCnf.DigIn_1_2.Text := WSTRING#'Ввідний пристрій: команда увімкн. лін. контактора';
   IO_Tags.InCnf.DigIn_1_3.Text := WSTRING#'Автомат трансформатора 9T1';
   IO_Tags.InCnf.DigIn_1_4.Text := WSTRING#'Автомат ремонтного освітлення';
   IO_Tags.InCnf.DigIn_1_5.Text := WSTRING#'Автомат власних потреб шафи';
   IO_Tags.InCnf.DigIn_1_6.Text := WSTRING#'Контроль обігріву шафи SU1';
   IO_Tags.InCnf.DigIn_2_0.Text := WSTRING#'Підйом: вгору, 1-ша швидк.';
   IO_Tags.InCnf.DigIn_2_1.Text := WSTRING#'Підйом: вниз, 1-ша швидк.';
   IO_Tags.InCnf.DigIn_2_2.Text := WSTRING#'Візок: вперед, 1-ша швидк.';
   IO_Tags.InCnf.DigIn_2_3.Text := WSTRING#'Візок: назад, 1-ша швидк.';
   IO_Tags.InCnf.DigIn_2_4.Text := WSTRING#'Кран: вліво, 1-ша швидк.';
   IO_Tags.InCnf.DigIn_2_5.Text := WSTRING#'Кран: вправо, 1-ша швидк.';
   IO_Tags.InCnf.DigIn_2_6.Text := WSTRING#'2-га швидкість';
   IO_Tags.InCnf.DigIn_2_7.Text := WSTRING#'Команда дзвінка';
   IO_Tags.InCnf.DigIn_3_2.Text := WSTRING#'Контроль роботи підйому';
   IO_Tags.InCnf.DigIn_3_3.Text := WSTRING#'Контроль зносу гальма підйому';
   IO_Tags.InCnf.DigIn_3_4.Text := WSTRING#'Підйом: дозв. роботи, РП роз’єдн.';
   IO_Tags.InCnf.DigIn_3_5.Text := WSTRING#'Кран: захист кіл гальм';
   IO_Tags.InCnf.DigIn_3_6.Text := WSTRING#'Кран: термозахист двигуна 4M1';
   IO_Tags.InCnf.DigIn_3_7.Text := WSTRING#'Кран: термозахист двигуна 4M2';
   IO_Tags.InCnf.DigIn_4_0.Text := WSTRING#'Підйом: термозахист гальм. резистора';
   IO_Tags.InCnf.DigIn_4_1.Text := WSTRING#'Підйом: дозв. норм. швидк., вгору';
   IO_Tags.InCnf.DigIn_4_2.Text := WSTRING#'Підйом: дозв. норм. швидк., вниз';
   IO_Tags.InCnf.DigIn_4_3.Text := WSTRING#'Підйом: дозв. руху вгору';
   IO_Tags.InCnf.DigIn_4_4.Text := WSTRING#'Підйом: дозв. руху вниз';
   IO_Tags.InCnf.DigIn_4_5.Text := WSTRING#'Підйом: перевантаження понад 115 %';
   IO_Tags.InCnf.DigIn_4_6.Text := WSTRING#'Підйом: слабина канатів';
   IO_Tags.InCnf.DigIn_4_7.Text := WSTRING#'Підйом: термозахист двигуна';
   IO_Tags.InCnf.DigIn_5_0.Text := WSTRING#'Підйом: КВ гальма 1YB1, розгальм.';
   IO_Tags.InCnf.DigIn_5_1.Text := WSTRING#'Підйом: КВ гальма 1YB1, загальм.';
   IO_Tags.InCnf.DigIn_5_3.Text := WSTRING#'Підйом: КВ гальма 1YB2, розгальм.';
   IO_Tags.InCnf.DigIn_5_4.Text := WSTRING#'Підйом: КВ гальма 1YB2, загальм.';
   IO_Tags.InCnf.DigIn_5_6.Text := WSTRING#'Підйом: захист випрямляча 1YB1';
   IO_Tags.InCnf.DigIn_5_7.Text := WSTRING#'Підйом: захист випрямляча 1YB2';
   IO_Tags.InCnf.DigIn_6_0.Text := WSTRING#'Візок: термозахист гальм. резистора';
   IO_Tags.InCnf.DigIn_6_1.Text := WSTRING#'Візок: дозв. норм. швидк., вперед';
   IO_Tags.InCnf.DigIn_6_2.Text := WSTRING#'Візок: дозв. руху вперед';
   IO_Tags.InCnf.DigIn_6_3.Text := WSTRING#'Візок: дозв. норм. швидк., назад';
   IO_Tags.InCnf.DigIn_6_4.Text := WSTRING#'Візок: дозв. руху назад';
   IO_Tags.InCnf.DigIn_6_5.Text := WSTRING#'Візок: дозв. роботи, РП роз’єдн.';
   IO_Tags.InCnf.DigIn_6_6.Text := WSTRING#'Візок: термозахист двигуна';
   IO_Tags.InCnf.DigIn_6_7.Text := WSTRING#'Дозв. роботи з обох боків колони';
   IO_Tags.InCnf.DigIn_7_0.Text := WSTRING#'Кран: термозахист резистора 4RT1';
   IO_Tags.InCnf.DigIn_7_1.Text := WSTRING#'Кран: термозахист резистора 4RT2';
   IO_Tags.InCnf.DigIn_7_2.Text := WSTRING#'Кран: дозв. норм. швидк., вліво';
   IO_Tags.InCnf.DigIn_7_3.Text := WSTRING#'Кран: дозв. норм. швидк., вправо';
   IO_Tags.InCnf.DigIn_7_4.Text := WSTRING#'Кран: дозв. руху вліво';
   IO_Tags.InCnf.DigIn_7_5.Text := WSTRING#'Кран: дозв. руху вправо';
   IO_Tags.InCnf.DigIn_7_6.Text := WSTRING#'Кран: дозв. роботи, РП роз’єдн. 4SQ41';
   IO_Tags.InCnf.DigIn_7_7.Text := WSTRING#'Кран: дозв. роботи, РП роз’єдн. 4SQ42';
   IO_Tags.InAnCfg.AnIn_0.Text := WSTRING#'Момент двигуна підйому';
   IO_Tags.OutCfg.DigOut_0_0.Text := WSTRING#'Увімкн. роб. гальма підйому';
   IO_Tags.OutCfg.DigOut_0_1.Text := WSTRING#'Увімкн. вбуд. гальма підйому';
   IO_Tags.OutCfg.DigOut_0_2.Text := WSTRING#'Увімкн. авар. гальма підйому';
   IO_Tags.OutCfg.DigOut_0_3.Text := WSTRING#'Увімкн. роб. гальма візка';
   IO_Tags.OutCfg.DigOut_0_4.Text := WSTRING#'Увімкн. роб. гальм крана';
   IO_Tags.OutCfg.DigOut_0_5.Text := WSTRING#'Дозв. увімкн. лін. контактора';
   IO_Tags.OutCfg.DigOut_0_6.Text := WSTRING#'Вимкн. лін. контактора';
   IO_Tags.OutCfg.DigOut_0_7.Text := WSTRING#'Увімкн. дзвінка';
   IO_Tags.OutCfg.DigOut_1_2.Text := WSTRING#'Лампа: готовність підйому';
   IO_Tags.OutCfg.DigOut_1_3.Text := WSTRING#'Лампа: готовність візка';
   IO_Tags.OutCfg.DigOut_1_4.Text := WSTRING#'Лампа: готовність крана';
   IO_Tags.OutCfg.DigOut_1_5.Text := WSTRING#'Лампа: лін. контактор увімкн.';
   IO_Tags.OutCfg.DigOut_1_6.Text := WSTRING#'Лампа: ввідна напруга не в нормі';
   IO_Tags.InAnCfg.AnIn_0.HIEng := 100.0;
   IO_Tags.InAnCfg.AnIn_0.LOEng := -100.0;
   IO_Tags.InAnCfg.AnIn_0.LORaw := -13824;
   IO_Tags.InAnCfg.AnIn_0.HIRaw := 13824;
   // IO_Tags.InCnf.DigIn_5_5 : Механізм підйому. Вимикачі кінцеві на гальмі 1YB2. Дозвіл роб. (MPP роз. з гальм.)
   // IO_Tags.InCnf.DigIn_5_2 : Механізм підйому. Вимикачі кінцеві на гальмі 1YB1. Товщ. гальм. накл. ОК
END_DATA_BLOCK

// folder: 100_InOut/InOut_DB

DATA_BLOCK "DB_AnIn_8"   // DB100
{ S7_Optimized_Access := 'TRUE' }
VERSION : 0.1
// stored: InstanceOfName FB_AnIn
"FB_AnIn"
BEGIN
END_DATA_BLOCK

DATA_BLOCK "DB_AnIn_10"   // DB101
{ S7_Optimized_Access := 'TRUE' }
VERSION : 0.1
// stored: InstanceOfName FB_AnIn
"FB_AnIn"
BEGIN
END_DATA_BLOCK

DATA_BLOCK "DB_AnIn_12"   // DB102
{ S7_Optimized_Access := 'TRUE' }
VERSION : 0.1
// stored: InstanceOfName FB_AnIn
"FB_AnIn"
BEGIN
END_DATA_BLOCK

DATA_BLOCK "DB_AnIn_14"   // DB103
{ S7_Optimized_Access := 'TRUE' }
VERSION : 0.1
// stored: InstanceOfName FB_AnIn
"FB_AnIn"
BEGIN
END_DATA_BLOCK

DATA_BLOCK "DB_AnIn_16"   // DB104
{ S7_Optimized_Access := 'TRUE' }
VERSION : 0.1
// stored: InstanceOfName FB_AnIn
"FB_AnIn"
BEGIN
END_DATA_BLOCK

DATA_BLOCK "DB_AnIn_18"   // DB105
{ S7_Optimized_Access := 'TRUE' }
VERSION : 0.1
// stored: InstanceOfName FB_AnIn
"FB_AnIn"
BEGIN
END_DATA_BLOCK

DATA_BLOCK "DB_AnIn_20"   // DB106
{ S7_Optimized_Access := 'TRUE' }
VERSION : 0.1
// stored: InstanceOfName FB_AnIn
"FB_AnIn"
BEGIN
END_DATA_BLOCK

DATA_BLOCK "DB_AnIn_22"   // DB107
{ S7_Optimized_Access := 'TRUE' }
VERSION : 0.1
// stored: InstanceOfName FB_AnIn
"FB_AnIn"
BEGIN
END_DATA_BLOCK

DATA_BLOCK "DB_DigIn_I0.0"   // DB108
{ S7_Optimized_Access := 'TRUE' }
VERSION : 0.1
// stored: InstanceOfName FB_DigIn
"FB_DigIn"
BEGIN
END_DATA_BLOCK

DATA_BLOCK "DB_DigIn_I0.1"   // DB109
{ S7_Optimized_Access := 'TRUE' }
VERSION : 0.1
// stored: InstanceOfName FB_DigIn
"FB_DigIn"
BEGIN
END_DATA_BLOCK

DATA_BLOCK "DB_DigIn_I0.2"   // DB110
{ S7_Optimized_Access := 'TRUE' }
VERSION : 0.1
// stored: InstanceOfName FB_DigIn
"FB_DigIn"
BEGIN
END_DATA_BLOCK

DATA_BLOCK "DB_DigIn_I0.3"   // DB111
{ S7_Optimized_Access := 'TRUE' }
VERSION : 0.1
// stored: InstanceOfName FB_DigIn
"FB_DigIn"
BEGIN
END_DATA_BLOCK

DATA_BLOCK "DB_DigIn_I0.4"   // DB112
{ S7_Optimized_Access := 'TRUE' }
VERSION : 0.1
// stored: InstanceOfName FB_DigIn
"FB_DigIn"
BEGIN
END_DATA_BLOCK

DATA_BLOCK "DB_DigIn_I0.5"   // DB113
{ S7_Optimized_Access := 'TRUE' }
VERSION : 0.1
// stored: InstanceOfName FB_DigIn
"FB_DigIn"
BEGIN
END_DATA_BLOCK

DATA_BLOCK "DB_DigIn_I0.6"   // DB114
{ S7_Optimized_Access := 'TRUE' }
VERSION : 0.1
// stored: InstanceOfName FB_DigIn
"FB_DigIn"
BEGIN
END_DATA_BLOCK

DATA_BLOCK "DB_DigIn_I0.7"   // DB115
{ S7_Optimized_Access := 'TRUE' }
VERSION : 0.1
// stored: InstanceOfName FB_DigIn
"FB_DigIn"
BEGIN
END_DATA_BLOCK

DATA_BLOCK "DB_DigIn_I1.0"   // DB116
{ S7_Optimized_Access := 'TRUE' }
VERSION : 0.1
// stored: InstanceOfName FB_DigIn
"FB_DigIn"
BEGIN
END_DATA_BLOCK

DATA_BLOCK "DB_DigIn_I1.1"   // DB117
{ S7_Optimized_Access := 'TRUE' }
VERSION : 0.1
// stored: InstanceOfName FB_DigIn
"FB_DigIn"
BEGIN
END_DATA_BLOCK

DATA_BLOCK "DB_DigIn_I1.2"   // DB118
{ S7_Optimized_Access := 'TRUE' }
VERSION : 0.1
// stored: InstanceOfName FB_DigIn
"FB_DigIn"
BEGIN
END_DATA_BLOCK

DATA_BLOCK "DB_DigIn_I1.3"   // DB119
{ S7_Optimized_Access := 'TRUE' }
VERSION : 0.1
// stored: InstanceOfName FB_DigIn
"FB_DigIn"
BEGIN
END_DATA_BLOCK

DATA_BLOCK "DB_DigIn_I1.4"   // DB120
{ S7_Optimized_Access := 'TRUE' }
VERSION : 0.1
// stored: InstanceOfName FB_DigIn
"FB_DigIn"
BEGIN
END_DATA_BLOCK

DATA_BLOCK "DB_DigIn_I1.5"   // DB121
{ S7_Optimized_Access := 'TRUE' }
VERSION : 0.1
// stored: InstanceOfName FB_DigIn
"FB_DigIn"
BEGIN
END_DATA_BLOCK

DATA_BLOCK "DB_DigIn_I1.6"   // DB122
{ S7_Optimized_Access := 'TRUE' }
VERSION : 0.1
// stored: InstanceOfName FB_DigIn
"FB_DigIn"
BEGIN
END_DATA_BLOCK

DATA_BLOCK "DB_DigIn_I1.7"   // DB123
{ S7_Optimized_Access := 'TRUE' }
VERSION : 0.1
// stored: InstanceOfName FB_DigIn
"FB_DigIn"
BEGIN
END_DATA_BLOCK

DATA_BLOCK "DB_DigIn_I2.0"   // DB124
{ S7_Optimized_Access := 'TRUE' }
VERSION : 0.1
// stored: InstanceOfName FB_DigIn
"FB_DigIn"
BEGIN
END_DATA_BLOCK

DATA_BLOCK "DB_DigIn_I2.1"   // DB125
{ S7_Optimized_Access := 'TRUE' }
VERSION : 0.1
// stored: InstanceOfName FB_DigIn
"FB_DigIn"
BEGIN
END_DATA_BLOCK

DATA_BLOCK "DB_DigIn_I2.2"   // DB126
{ S7_Optimized_Access := 'TRUE' }
VERSION : 0.1
// stored: InstanceOfName FB_DigIn
"FB_DigIn"
BEGIN
END_DATA_BLOCK

DATA_BLOCK "DB_DigIn_I2.3"   // DB127
{ S7_Optimized_Access := 'TRUE' }
VERSION : 0.1
// stored: InstanceOfName FB_DigIn
"FB_DigIn"
BEGIN
END_DATA_BLOCK

DATA_BLOCK "DB_DigIn_I2.4"   // DB128
{ S7_Optimized_Access := 'TRUE' }
VERSION : 0.1
// stored: InstanceOfName FB_DigIn
"FB_DigIn"
BEGIN
END_DATA_BLOCK

DATA_BLOCK "DB_DigIn_I2.5"   // DB129
{ S7_Optimized_Access := 'TRUE' }
VERSION : 0.1
// stored: InstanceOfName FB_DigIn
"FB_DigIn"
BEGIN
END_DATA_BLOCK

DATA_BLOCK "DB_DigIn_I2.6"   // DB130
{ S7_Optimized_Access := 'TRUE' }
VERSION : 0.1
// stored: InstanceOfName FB_DigIn
"FB_DigIn"
BEGIN
END_DATA_BLOCK

DATA_BLOCK "DB_DigIn_I2.7"   // DB131
{ S7_Optimized_Access := 'TRUE' }
VERSION : 0.1
// stored: InstanceOfName FB_DigIn
"FB_DigIn"
BEGIN
END_DATA_BLOCK

DATA_BLOCK "DB_DigIn_I3.0"   // DB132
{ S7_Optimized_Access := 'TRUE' }
VERSION : 0.1
// stored: InstanceOfName FB_DigIn
"FB_DigIn"
BEGIN
END_DATA_BLOCK

DATA_BLOCK "DB_DigIn_I3.1"   // DB133
{ S7_Optimized_Access := 'TRUE' }
VERSION : 0.1
// stored: InstanceOfName FB_DigIn
"FB_DigIn"
BEGIN
END_DATA_BLOCK

DATA_BLOCK "DB_DigIn_I3.2"   // DB134
{ S7_Optimized_Access := 'TRUE' }
VERSION : 0.1
// stored: InstanceOfName FB_DigIn
"FB_DigIn"
BEGIN
END_DATA_BLOCK

DATA_BLOCK "DB_DigIn_I3.3"   // DB135
{ S7_Optimized_Access := 'TRUE' }
VERSION : 0.1
// stored: InstanceOfName FB_DigIn
"FB_DigIn"
BEGIN
END_DATA_BLOCK

DATA_BLOCK "DB_DigIn_I3.4"   // DB136
{ S7_Optimized_Access := 'TRUE' }
VERSION : 0.1
// stored: InstanceOfName FB_DigIn
"FB_DigIn"
BEGIN
END_DATA_BLOCK

DATA_BLOCK "DB_DigIn_I3.5"   // DB137
{ S7_Optimized_Access := 'TRUE' }
VERSION : 0.1
// stored: InstanceOfName FB_DigIn
"FB_DigIn"
BEGIN
END_DATA_BLOCK

